KUKA KRL program: MyProgram_167().src

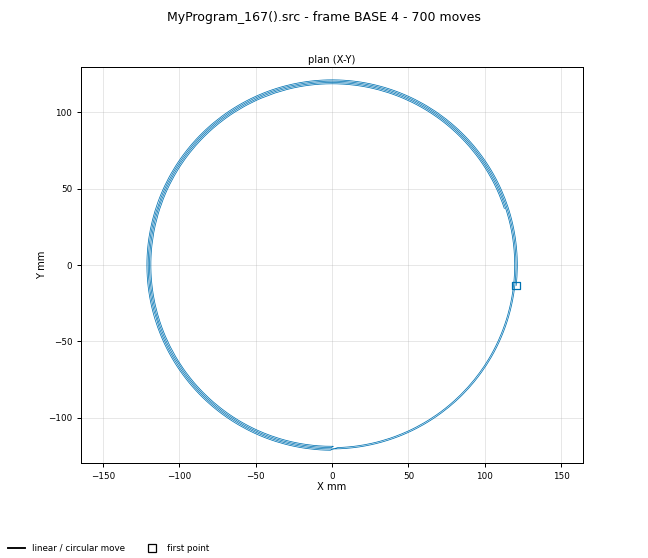
[picture p0: tool path of MyProgram_167().src in frame BASE 4, 700 of 700 moves have a stored position in this frame; points joined in program order, loops and branches not executed]
&ACCESS RVP
&REL 1
&PARAM TEMPLATE = C:\KRC\Roboter\Template\vorgabe
&PARAM EDITMASK = *
DEF MyProgram_167()
; ---- Setting reference (Base) ----
$BASE = BASE_DATA[4]

; --------------------------
; ---- Setting tool (TCP) ----
$TOOL = TOOL_DATA[3]
; --------------------------

$VEL.CP = VEL_APROX_PRINT
Startdeposition()
$VEL.CP = VEL_PRINT
LIN {X 120.5088,Y -13.3642,Z 126,A -9.8164,B 24.9507,C -1.6218,E1 25.1589,E2 455.9216} C_DIS
LIN {X 120.8004,Y -10.4027,Z 126,A -8.4201,B 24.9505,C -1.6259,E1 25.1593,E2 454.5239} C_DIS
LIN {X 121.0193,Y -7.435,Z 126,A -7.0235,B 24.9502,C -1.63,E1 25.1595,E2 453.1259} C_DIS
LIN {X 121.1789,Y -4.022,Z 126,A -5.6063,B 24.9505,C -1.6254,E1 25.1597,E2 451.728} C_DIS
LIN {X 121.2384,Y -1.4879,Z 126,A -4.2539,B 24.9498,C -1.6371,E1 25.1597,E2 450.3561} C_DIS
LIN {X 121.2384,Y 1.4879,Z 126,A -2.834,B 24.9495,C -1.6424,E1 25.1597,E2 448.9323} C_DIS
LIN {X 121.1654,Y 4.4628,Z 126,A -1.4376,B 24.9492,C -1.6465,E1 25.1597,E2 447.5345} C_DIS
LIN {X 121.0193,Y 7.435,Z 126,A -0.0409,B 24.9489,C -1.6506,E1 25.1594,E2 446.1364} C_DIS
LIN {X 120.7573,Y 10.8703,Z 126,A 1.6055,B 24.9486,C -1.6568,E1 25.159,E2 444.4851} C_DIS
LIN {X 120.3357,Y 14.842,Z 126,A 3.4507,B 24.9483,C -1.6607,E1 25.1585,E2 442.6415} C_DIS
LIN {X 119.9352,Y 17.7907,Z 126,A 4.8473,B 24.9481,C -1.6648,E1 25.1579,E2 441.2437} C_DIS
LIN {X 119.4625,Y 20.7287,Z 126,A 6.2442,B 24.9478,C -1.6688,E1 25.1573,E2 439.8455} C_DIS
LIN {X 118.9178,Y 23.6542,Z 126,A 7.6407,B 24.9476,C -1.6728,E1 25.1565,E2 438.4477} C_DIS
LIN {X 118.3015,Y 26.5655,Z 126,A 9.0377,B 24.9473,C -1.6767,E1 25.1557,E2 437.0495} C_DIS
LIN {X 117.6139,Y 29.4607,Z 126,A 10.4346,B 24.9471,C -1.6807,E1 25.1548,E2 435.6514} C_DIS
LIN {X 116.8555,Y 32.3383,Z 126,A 11.8317,B 24.9468,C -1.6846,E1 25.1537,E2 434.2532} C_DIS
LIN {X 116.0266,Y 35.1963,Z 126,A 13.2287,B 24.9466,C -1.6884,E1 25.1526,E2 432.855} C_DIS
LIN {X 115.1279,Y 38.0331,Z 126,A 14.6257,B 24.9463,C -1.6923,E1 25.1514,E2 431.4568} C_DIS
LIN {X 114.0244,Y 41.2185,Z 126,A 16.0417,B 24.9466,C -1.6883,E1 25.1501,E2 430.0583} C_DIS
LIN {X 113.1231,Y 43.6364,Z 126,A 17.5207,B 24.9455,C -1.7048,E1 25.1486,E2 428.5485} C_DIS
LIN {X 111.7931,Y 46.9333,Z 126,A 18.8451,B 24.9463,C -1.6921,E1 25.1473,E2 427.2613} C_DIS
LIN {X 110.8457,Y 49.1345,Z 126,A 20.2154,B 24.9454,C -1.7072,E1 25.1457,E2 425.863} C_DIS
LIN {X 109.6065,Y 51.84,Z 126,A 21.613,B 24.9451,C -1.7108,E1 25.1441,E2 424.4644} C_DIS
LIN {X 108.3012,Y 54.5143,Z 126,A 23.0108,B 24.9449,C -1.7144,E1 25.1423,E2 423.0656} C_DIS
LIN {X 106.9308,Y 57.1557,Z 126,A 24.4089,B 24.9447,C -1.7179,E1 25.1405,E2 421.6666} C_DIS
LIN {X 105.4959,Y 59.7627,Z 126,A 25.9523,B 24.944,C -1.7286,E1 25.1384,E2 420.106} C_DIS
LIN {X 103.9975,Y 62.3337,Z 126,A 27.2051,B 24.9442,C -1.7248,E1 25.1366,E2 418.8687} C_DIS
LIN {X 102.4364,Y 64.8671,Z 126,A 28.6034,B 24.944,C -1.7281,E1 25.1345,E2 417.4696} C_DIS
LIN {X 100.8136,Y 67.3615,Z 126,A 30.1196,B 24.9434,C -1.7372,E1 25.1322,E2 415.9394} C_DIS
LIN {X 98.2659,Y 71.0265,Z 126,A 32.0998,B 24.9435,C -1.7363,E1 25.129,E2 413.9712} C_DIS
LIN {X 96.4932,Y 73.4167,Z 126,A 33.4984,B 24.9433,C -1.7394,E1 25.1267,E2 412.5719} C_DIS
LIN {X 94.6625,Y 75.7627,Z 126,A 34.8975,B 24.9431,C -1.7425,E1 25.1242,E2 411.172} C_DIS
LIN {X 92.7746,Y 78.063,Z 126,A 36.2965,B 24.9429,C -1.7455,E1 25.1217,E2 409.7723} C_DIS
LIN {X 90.8309,Y 80.3163,Z 126,A 37.6959,B 24.9427,C -1.7484,E1 25.1192,E2 408.3724} C_DIS
LIN {X 88.8325,Y 82.5212,Z 126,A 39.0953,B 24.9425,C -1.7513,E1 25.1165,E2 406.9724} C_DIS
LIN {X 86.7806,Y 84.6764,Z 126,A 40.4951,B 24.9423,C -1.7541,E1 25.1138,E2 405.572} C_DIS
LIN {X 84.6764,Y 86.7806,Z 126,A 41.8949,B 24.9422,C -1.7568,E1 25.111,E2 404.1717} C_DIS
LIN {X 82.5212,Y 88.8325,Z 126,A 43.2949,B 24.942,C -1.7594,E1 25.1082,E2 402.7712} C_DIS
LIN {X 80.3163,Y 90.8309,Z 126,A 44.8186,B 24.9414,C -1.768,E1 25.105,E2 401.2334} C_DIS
LIN {X 77.6174,Y 93.1449,Z 126,A 46.368,B 24.9416,C -1.7649,E1 25.1017,E2 399.6971} C_DIS
LIN {X 74.5953,Y 95.585,Z 126,A 48.1962,B 24.9414,C -1.768,E1 25.0977,E2 397.8685} C_DIS
LIN {X 72.0735,Y 97.4993,Z 126,A 49.6061,B 24.9415,C -1.7665,E1 25.0946,E2 396.4672} C_DIS
LIN {X 69.8153,Y 99.1301,Z 126,A 50.9982,B 24.9411,C -1.7725,E1 25.0914,E2 395.0659} C_DIS
LIN {X 67.3615,Y 100.8136,Z 126,A 52.3996,B 24.941,C -1.7746,E1 25.0881,E2 393.6643} C_DIS
LIN {X 64.7375,Y 102.5174,Z 126,A 53.8079,B 24.941,C -1.7736,E1 25.0849,E2 392.2629} C_DIS
LIN {X 62.3337,Y 103.9975,Z 126,A 55.2026,B 24.9407,C -1.7785,E1 25.0815,E2 390.8609} C_DIS
LIN {X 59.7627,Y 105.4959,Z 126,A 56.6046,B 24.9406,C -1.7804,E1 25.0781,E2 389.4587} C_DIS
LIN {X 56.9784,Y 107.0241,Z 126,A 58.0159,B 24.9407,C -1.7782,E1 25.0747,E2 388.0567} C_DIS
LIN {X 54.5143,Y 108.3012,Z 126,A 59.409,B 24.9404,C -1.7838,E1 25.0712,E2 386.6541} C_DIS
LIN {X 51.84,Y 109.6065,Z 126,A 60.8116,B 24.9403,C -1.7853,E1 25.0676,E2 385.2515} C_DIS
LIN {X 48.6786,Y 111.0444,Z 126,A 62.4707,B 24.9401,C -1.7881,E1 25.0634,E2 383.59} C_DIS
LIN {X 45.0213,Y 112.5791,Z 126,A 64.3189,B 24.9401,C -1.7888,E1 25.0586,E2 381.7443} C_DIS
LIN {X 42.2449,Y 113.65,Z 126,A 65.7222,B 24.9399,C -1.79,E1 25.055,E2 380.3412} C_DIS
LIN {X 39.4431,Y 114.6525,Z 126,A 67.1257,B 24.9399,C -1.7912,E1 25.0513,E2 378.9378} C_DIS
LIN {X 36.6175,Y 115.586,Z 126,A 68.5295,B 24.9398,C -1.7922,E1 25.0476,E2 377.5342} C_DIS
LIN {X 33.7698,Y 116.4498,Z 126,A 69.9336,B 24.9398,C -1.7931,E1 25.0438,E2 376.1303} C_DIS
LIN {X 30.9018,Y 117.2435,Z 126,A 71.3378,B 24.9397,C -1.794,E1 25.04,E2 374.7263} C_DIS
LIN {X 28.0152,Y 117.9666,Z 126,A 72.7421,B 24.9397,C -1.7947,E1 25.0362,E2 373.3224} C_DIS
LIN {X 25.1117,Y 118.6186,Z 126,A 74.1469,B 24.9396,C -1.7953,E1 25.0324,E2 371.9178} C_DIS
LIN {X 22.1931,Y 119.1991,Z 126,A 75.7244,B 24.939,C -1.804,E1 25.028,E2 370.3218} C_DIS
LIN {X 19.2612,Y 119.7078,Z 126,A 76.9573,B 24.9395,C -1.7963,E1 25.0246,E2 369.1082} C_DIS
LIN {X 16.3176,Y 120.1445,Z 126,A 78.3627,B 24.9395,C -1.7967,E1 25.0208,E2 367.7033} C_DIS
LIN {X 13.3642,Y 120.5088,Z 126,A 79.7685,B 24.9395,C -1.7969,E1 25.0169,E2 366.298} C_DIS
LIN {X 10.4027,Y 120.8004,Z 126,A 81.1742,B 24.9395,C -1.797,E1 25.013,E2 364.8928} C_DIS
LIN {X 7.435,Y 121.0193,Z 126,A 82.5805,B 24.9395,C -1.797,E1 25.009,E2 363.4871} C_DIS
LIN {X 4.4628,Y 121.1654,Z 126,A 84.1576,B 24.9389,C -1.8049,E1 25.0046,E2 361.8918} C_DIS
LIN {X 0.8202,Y 121.2425,Z 126,A 85.687,B 24.9396,C -1.7958,E1 25.0004,E2 360.3842} C_DIS
LIN {X -2.9756,Y 121.211,Z 126,A 87.5041,B 24.9396,C -1.7964,E1 24.9953,E2 358.5656} C_DIS
LIN {X -5.9493,Y 121.1015,Z 126,A 88.9114,B 24.9396,C -1.7959,E1 24.9914,E2 357.159} C_DIS
LIN {X -8.9195,Y 120.919,Z 126,A 90.319,B 24.9396,C -1.7954,E1 24.9875,E2 355.7522} C_DIS
LIN {X -11.8843,Y 120.6637,Z 126,A 91.7265,B 24.9396,C -1.7948,E1 24.9835,E2 354.3454} C_DIS
LIN {X -14.842,Y 120.3357,Z 126,A 93.1491,B 24.9396,C -1.7948,E1 24.9796,E2 352.9221} C_DIS
LIN {X -17.7907,Y 119.9352,Z 126,A 94.5427,B 24.9397,C -1.7932,E1 24.9758,E2 351.5309} C_DIS
LIN {X -20.7287,Y 119.4625,Z 126,A 95.9513,B 24.9397,C -1.7923,E1 24.9719,E2 350.1231} C_DIS
LIN {X -23.6542,Y 118.9178,Z 126,A 97.3599,B 24.9399,C -1.7913,E1 24.968,E2 348.7153} C_DIS
LIN {X -26.5655,Y 118.3015,Z 126,A 98.9351,B 24.9394,C -1.7977,E1 24.9637,E2 347.123} C_DIS
LIN {X -30.9018,Y 117.2435,Z 126,A 100.8828,B 24.9401,C -1.7883,E1 24.9585,E2 345.1949} C_DIS
LIN {X -33.7698,Y 116.4498,Z 126,A 102.2921,B 24.9401,C -1.7869,E1 24.9547,E2 343.7865} C_DIS
LIN {X -36.6175,Y 115.586,Z 126,A 103.7017,B 24.9403,C -1.7854,E1 24.9509,E2 342.378} C_DIS
LIN {X -39.4431,Y 114.6525,Z 126,A 105.1119,B 24.9403,C -1.7839,E1 24.9472,E2 340.9688} C_DIS
LIN {X -42.2449,Y 113.65,Z 126,A 106.5502,B 24.9403,C -1.7835,E1 24.9434,E2 339.5285} C_DIS
LIN {X -45.0213,Y 112.5791,Z 126,A 107.9324,B 24.9406,C -1.7805,E1 24.9398,E2 338.1506} C_DIS
LIN {X -47.7706,Y 111.4403,Z 126,A 109.3428,B 24.9407,C -1.7786,E1 24.9362,E2 336.7413} C_DIS
LIN {X -50.4911,Y 110.2344,Z 126,A 110.7536,B 24.9408,C -1.7767,E1 24.9326,E2 335.3316} C_DIS
LIN {X -53.1811,Y 108.9621,Z 126,A 112.1649,B 24.941,C -1.7747,E1 24.9291,E2 333.9215} C_DIS
LIN {X -55.8619,Y 107.6121,Z 126,A 113.7461,B 24.9406,C -1.7796,E1 24.9251,E2 332.3244} C_DIS
LIN {X -58.9695,Y 105.9388,Z 126,A 115.2623,B 24.9413,C -1.77,E1 24.9214,E2 330.8267} C_DIS
LIN {X -62.3337,Y 103.9975,Z 126,A 117.1167,B 24.9415,C -1.7674,E1 24.917,E2 328.9728} C_DIS
LIN {X -64.8671,Y 102.4364,Z 126,A 118.5171,B 24.9416,C -1.7645,E1 24.9137,E2 327.5749} C_DIS
LIN {X -67.3615,Y 100.8136,Z 126,A 119.9293,B 24.9418,C -1.762,E1 24.9104,E2 326.164} C_DIS
LIN {X -69.8153,Y 99.1301,Z 126,A 121.3416,B 24.942,C -1.7594,E1 24.9071,E2 324.753} C_DIS
LIN {X -72.2271,Y 97.3869,Z 126,A 122.7544,B 24.9422,C -1.7568,E1 24.9039,E2 323.3415} C_DIS
LIN {X -75.0019,Y 95.2637,Z 126,A 124.1911,B 24.943,C -1.7438,E1 24.9008,E2 321.9303} C_DIS
LIN {X -76.9186,Y 93.7256,Z 126,A 125.5798,B 24.9425,C -1.7512,E1 24.8978,E2 320.5189} C_DIS
LIN {X -79.1956,Y 91.8097,Z 126,A 126.9929,B 24.9427,C -1.7483,E1 24.8948,E2 319.1072} C_DIS
LIN {X -81.4249,Y 89.8385,Z 126,A 128.4063,B 24.9429,C -1.7454,E1 24.8918,E2 317.6951} C_DIS
LIN {X -83.6051,Y 87.8132,Z 126,A 129.9755,B 24.9427,C -1.7492,E1 24.8886,E2 316.1105} C_DIS
LIN {X -86.8025,Y 84.6536,Z 126,A 131.9416,B 24.9435,C -1.737,E1 24.8848,E2 314.1649} C_DIS
LIN {X -88.8325,Y 82.5212,Z 126,A 133.3537,B 24.9436,C -1.7344,E1 24.8821,E2 312.7528} C_DIS
LIN {X -90.8309,Y 80.3163,Z 126,A 134.768,B 24.9438,C -1.7312,E1 24.8794,E2 311.34} C_DIS
LIN {X -92.7964,Y 78.0368,Z 126,A 136.1837,B 24.9441,C -1.7272,E1 24.8769,E2 309.9273} C_DIS
LIN {X -94.9311,Y 75.4227,Z 126,A 137.8426,B 24.9441,C -1.7258,E1 24.874,E2 308.2641} C_DIS
LIN {X -97.3869,Y 72.2271,Z 126,A 139.7182,B 24.9446,C -1.7193,E1 24.8708,E2 306.3951} C_DIS
LIN {X -99.1301,Y 69.8153,Z 126,A 141.1328,B 24.9448,C -1.7157,E1 24.8685,E2 304.9819} C_DIS
LIN {X -100.8136,Y 67.3615,Z 126,A 142.5475,B 24.9451,C -1.7121,E1 24.8663,E2 303.5687} C_DIS
LIN {X -102.4364,Y 64.8671,Z 126,A 143.9623,B 24.9453,C -1.7085,E1 24.8642,E2 302.1554} C_DIS
LIN {X -104.1525,Y 62.0714,Z 126,A 145.3916,B 24.9459,C -1.6988,E1 24.8621,E2 300.7419} C_DIS
LIN {X -105.4959,Y 59.7627,Z 126,A 146.7923,B 24.9458,C -1.7011,E1 24.8602,E2 299.3285} C_DIS
LIN {X -106.9308,Y 57.1557,Z 126,A 148.2076,B 24.946,C -1.6973,E1 24.8583,E2 297.9147} C_DIS
LIN {X -108.3095,Y 54.4976,Z 126,A 149.6237,B 24.9463,C -1.6931,E1 24.8565,E2 296.501} C_DIS
LIN {X -109.6065,Y 51.84,Z 126,A 151.0383,B 24.9465,C -1.6896,E1 24.8548,E2 295.0871} C_DIS
LIN {X -110.8457,Y 49.1345,Z 126,A 152.4539,B 24.9467,C -1.6857,E1 24.8532,E2 293.6731} C_DIS
LIN {X -112.0181,Y 46.3994,Z 126,A 153.8695,B 24.947,C -1.6818,E1 24.8516,E2 292.259} C_DIS
LIN {X -113.1231,Y 43.6364,Z 126,A 155.2851,B 24.9472,C -1.6778,E1 24.8502,E2 290.8449} C_DIS
LIN {X -114.1599,Y 40.8471,Z 126,A 156.7007,B 24.9475,C -1.6738,E1 24.8488,E2 289.4308} C_DIS
LIN {X -115.2699,Y 37.5944,Z 126,A 158.1384,B 24.9483,C -1.6607,E1 24.8476,E2 288.0162} C_DIS
LIN {X -116.0266,Y 35.1963,Z 126,A 159.6235,B 24.9478,C -1.6696,E1 24.8463,E2 286.5012} C_DIS
LIN {X -117.0066,Y 31.7789,Z 126,A 160.9754,B 24.949,C -1.6502,E1 24.8453,E2 285.1878} C_DIS
LIN {X -117.6139,Y 29.4607,Z 126,A 162.4636,B 24.9483,C -1.6618,E1 24.8443,E2 283.6633} C_DIS
LIN {X -118.4249,Y 25.9994,Z 126,A 163.8076,B 24.9495,C -1.642,E1 24.8435,E2 282.3586} C_DIS
LIN {X -118.9626,Y 23.4216,Z 126,A 165.2076,B 24.9493,C -1.6446,E1 24.8427,E2 280.9441} C_DIS
LIN {X -119.4625,Y 20.7287,Z 126,A 166.6128,B 24.9493,C -1.6451,E1 24.842,E2 279.5293} C_DIS
LIN {X -119.9352,Y 17.7907,Z 126,A 168.0287,B 24.9495,C -1.641,E1 24.8414,E2 278.1149} C_DIS
LIN {X -120.3357,Y 14.842,Z 126,A 169.4448,B 24.9498,C -1.6368,E1 24.8409,E2 276.7003} C_DIS
LIN {X -120.6637,Y 11.8843,Z 126,A 170.8611,B 24.9501,C -1.6327,E1 24.8405,E2 275.2854} C_DIS
LIN {X -120.919,Y 8.9195,Z 126,A 172.2771,B 24.9503,C -1.6285,E1 24.8401,E2 273.8708} C_DIS
LIN {X -121.1015,Y 5.9493,Z 126,A 173.6934,B 24.9506,C -1.6243,E1 24.8399,E2 272.4559} C_DIS
LIN {X -121.211,Y 2.9756,Z 126,A 175.1095,B 24.9508,C -1.6201,E1 24.8399,E2 271.0413} C_DIS
LIN {X -121.2455,Y -0.4051,Z 126,A 176.7824,B 24.9509,C -1.6182,E1 24.8398,E2 269.3629} C_DIS
LIN {X -121.1654,Y -4.4628,Z 126,A 178.6495,B 24.9514,C -1.6097,E1 24.8399,E2 267.5048} C_DIS
LIN {X -121.013,Y -7.5284,Z 126,A -179.7941,B 24.9514,C -1.6097,E1 24.8402,E2 265.9393} C_DIS
LIN {X -120.6637,Y -11.8843,Z 126,A -177.8103,B 24.9521,C -1.5994,E1 24.8407,E2 263.9679} C_DIS
LIN {X -120.3357,Y -14.842,Z 126,A -176.3942,B 24.9523,C -1.5953,E1 24.8411,E2 262.5531} C_DIS
LIN {X -119.9352,Y -17.7907,Z 126,A -174.9784,B 24.9526,C -1.5912,E1 24.8417,E2 261.1386} C_DIS
LIN {X -119.4625,Y -20.7287,Z 126,A -173.5624,B 24.9528,C -1.5872,E1 24.8423,E2 259.7238} C_DIS
LIN {X -118.9178,Y -23.6542,Z 126,A -172.1466,B 24.953,C -1.5831,E1 24.8431,E2 258.3092} C_DIS
LIN {X -118.3015,Y -26.5655,Z 126,A -170.7307,B 24.9533,C -1.5791,E1 24.8439,E2 256.8945} C_DIS
LIN {X -117.6139,Y -29.4607,Z 126,A -169.3152,B 24.9535,C -1.5752,E1 24.8449,E2 255.4803} C_DIS
LIN {X -116.8555,Y -32.3383,Z 126,A -167.8998,B 24.9537,C -1.5712,E1 24.8459,E2 254.0661} C_DIS
LIN {X -116.0266,Y -35.1963,Z 126,A -166.4841,B 24.954,C -1.5673,E1 24.847,E2 252.6515} C_DIS
LIN {X -115.0484,Y -38.2691,Z 126,A -164.8855,B 24.954,C -1.5659,E1 24.8484,E2 251.047} C_DIS
LIN {X -114.1599,Y -40.8471,Z 126,A -163.6533,B 24.9544,C -1.5596,E1 24.8496,E2 249.823} C_DIS
LIN {X -113.0904,Y -43.7196,Z 126,A -162.2341,B 24.9548,C -1.554,E1 24.8509,E2 248.409} C_DIS
LIN {X -112.0181,Y -46.3994,Z 126,A -160.8227,B 24.9548,C -1.5521,E1 24.8524,E2 246.9945} C_DIS
LIN {X -110.8457,Y -49.1345,Z 126,A -159.4081,B 24.9551,C -1.5483,E1 24.854,E2 245.5809} C_DIS
LIN {X -109.6065,Y -51.84,Z 126,A -157.993,B 24.9553,C -1.5447,E1 24.8557,E2 244.1668} C_DIS
LIN {X -108.3012,Y -54.5143,Z 126,A -156.5784,B 24.9555,C -1.5411,E1 24.8574,E2 242.7531} C_DIS
LIN {X -106.9308,Y -57.1557,Z 126,A -155.1021,B 24.9555,C -1.5402,E1 24.8594,E2 241.271} C_DIS
LIN {X -105.2072,Y -60.2651,Z 126,A -153.4738,B 24.9559,C -1.5334,E1 24.8616,E2 239.6504} C_DIS
LIN {X -103.2247,Y -63.6052,Z 126,A -151.6275,B 24.9562,C -1.5289,E1 24.8643,E2 237.8053} C_DIS
LIN {X -101.6327,Y -66.1193,Z 126,A -150.2134,B 24.9564,C -1.5256,E1 24.8664,E2 236.3921} C_DIS
LIN {X -99.8332,Y -68.8039,Z 126,A -148.5835,B 24.9564,C -1.5262,E1 24.869,E2 234.7526} C_DIS
LIN {X -97.9236,Y -71.494,Z 126,A -147.1102,B 24.9568,C -1.5185,E1 24.8713,E2 233.2904} C_DIS
LIN {X -95.5851,Y -74.5953,Z 126,A -145.2649,B 24.957,C -1.5144,E1 24.8745,E2 231.4462} C_DIS
LIN {X -93.7256,Y -76.9186,Z 126,A -143.8516,B 24.9572,C -1.5113,E1 24.877,E2 230.0335} C_DIS
LIN {X -91.8097,Y -79.1956,Z 126,A -142.4382,B 24.9574,C -1.5084,E1 24.8795,E2 228.6208} C_DIS
LIN {X -89.8385,Y -81.4249,Z 126,A -140.9105,B 24.9573,C -1.5106,E1 24.8824,E2 227.081} C_DIS
LIN {X -86.7806,Y -84.6764,Z 126,A -138.9054,B 24.9578,C -1.5013,E1 24.8862,E2 225.0894} C_DIS
LIN {X -84.6764,Y -86.7806,Z 126,A -137.4929,B 24.9579,C -1.4985,E1 24.889,E2 223.6774} C_DIS
LIN {X -82.5212,Y -88.8325,Z 126,A -135.9178,B 24.9577,C -1.5032,E1 24.8923,E2 222.0848} C_DIS
LIN {X -80.3163,Y -90.8309,Z 126,A -134.6681,B 24.9582,C -1.4933,E1 24.8949,E2 220.8536} C_DIS
LIN {X -78.063,Y -92.7746,Z 126,A -133.2263,B 24.9582,C -1.4922,E1 24.8979,E2 219.4088} C_DIS
LIN {X -75.7627,Y -94.6625,Z 126,A -131.7323,B 24.9582,C -1.4935,E1 24.9012,E2 217.9062} C_DIS
LIN {X -73.4167,Y -96.4932,Z 126,A -130.4327,B 24.9586,C -1.4862,E1 24.904,E2 216.6193} C_DIS
LIN {X -71.0265,Y -98.2659,Z 126,A -129.0209,B 24.9587,C -1.484,E1 24.9072,E2 215.2078} C_DIS
LIN {X -68.5936,Y -99.9794,Z 126,A -127.5133,B 24.9587,C -1.4862,E1 24.9107,E2 213.6898} C_DIS
LIN {X -66.1193,Y -101.6327,Z 126,A -126.1986,B 24.959,C -1.4798,E1 24.9137,E2 212.3859} C_DIS
LIN {X -63.6052,Y -103.2247,Z 126,A -124.7876,B 24.959,C -1.4778,E1 24.9171,E2 210.9752} C_DIS
LIN {X -61.0528,Y -104.7546,Z 126,A -123.2908,B 24.959,C -1.4799,E1 24.9207,E2 209.4689} C_DIS
LIN {X -57.9543,Y -106.4976,Z 126,A -121.9393,B 24.9599,C -1.4627,E1 24.9239,E2 208.1545} C_DIS
LIN {X -55.8392,Y -107.6241,Z 126,A -120.4877,B 24.9592,C -1.4757,E1 24.9276,E2 206.6679} C_DIS
LIN {X -53.1811,Y -108.9621,Z 126,A -118.9981,B 24.9591,C -1.4777,E1 24.9313,E2 205.1695} C_DIS
LIN {X -50.4911,Y -110.2344,Z 126,A -117.7365,B 24.9595,C -1.4695,E1 24.9345,E2 203.9244} C_DIS
LIN {X -47.7706,Y -111.4403,Z 126,A -116.3273,B 24.9596,C -1.4681,E1 24.9381,E2 202.5153} C_DIS
LIN {X -45.0213,Y -112.5791,Z 126,A -114.9176,B 24.9596,C -1.4668,E1 24.9418,E2 201.1055} C_DIS
LIN {X -42.2449,Y -113.65,Z 126,A -113.5087,B 24.9598,C -1.4656,E1 24.9454,E2 199.6964} C_DIS
LIN {X -39.4431,Y -114.6525,Z 126,A -112.0997,B 24.9598,C -1.4645,E1 24.9491,E2 198.2873} C_DIS
LIN {X -36.6175,Y -115.586,Z 126,A -110.6913,B 24.9598,C -1.4635,E1 24.9529,E2 196.8787} C_DIS
LIN {X -33.4991,Y -116.5265,Z 126,A -109.0639,B 24.9598,C -1.4665,E1 24.9573,E2 195.2415} C_DIS
LIN {X -30.9018,Y -117.2435,Z 126,A -107.8747,B 24.96,C -1.4618,E1 24.9605,E2 194.0616} C_DIS
LIN {X -28.0152,Y -117.9666,Z 126,A -106.4671,B 24.96,C -1.4611,E1 24.9643,E2 192.6537} C_DIS
LIN {X -25.1117,Y -118.6186,Z 126,A -105.0151,B 24.96,C -1.4626,E1 24.9683,E2 191.1965} C_DIS
LIN {X -22.1931,Y -119.1991,Z 126,A -103.6519,B 24.96,C -1.46,E1 24.972,E2 189.8378} C_DIS
LIN {X -19.2612,Y -119.7078,Z 126,A -102.2445,B 24.96,C -1.4596,E1 24.9759,E2 188.43} C_DIS
LIN {X -16.3176,Y -120.1445,Z 126,A -100.8377,B 24.9601,C -1.4593,E1 24.9798,E2 187.0228} C_DIS
LIN {X -12.8412,Y -120.5635,Z 126,A -99.3639,B 24.9606,C -1.4507,E1 24.9838,E2 185.5686} C_DIS
LIN {X -10.4027,Y -120.8004,Z 126,A -98.0247,B 24.9601,C -1.4591,E1 24.9876,E2 184.2088} C_DIS
LIN {X -7.435,Y -121.0193,Z 126,A -96.6184,B 24.9601,C -1.4591,E1 24.9915,E2 182.8019} C_DIS
LIN {X -4.4628,Y -121.1654,Z 126,A -95.2124,B 24.9601,C -1.4592,E1 24.9954,E2 181.3953} C_DIS
LIN {X -1.1524,Y -121.2404,Z 126,A -93.5793,B 24.9599,C -1.4627,E1 25,E2 179.7537} C_DIS
LIN {X -1.1524,Y -121.2404,Z 126,A -93.5793,B 24.9599,C -1.4627,E1 25,E2 179.7537} C_DIS
Enddeposition()
LIN {X 0.8412,Y -120.3739,Z 126,A -92.3537,B 24.9583,C -1.4914,E1 25.0036,E2 178.4603} C_DIS
Startdeposition()
$VEL.CP = VEL_PRINT
LIN {X -0.5989,Y -120.3841,Z 126,A -94.8852,B 24.963,C -1.4054,E1 24.996,E2 181.1955} C_DIS
LIN {X -6.0161,Y -120.2368,Z 126,A -96.5858,B 24.9609,C -1.4454,E1 24.9915,E2 182.8019} C_DIS
LIN {X -10.8702,Y -119.8939,Z 126,A -98.8361,B 24.9607,C -1.4484,E1 24.9853,E2 185.0458} C_DIS
LIN {X -17.8185,Y -119.061,Z 126,A -102.2139,B 24.9607,C -1.4467,E1 24.9759,E2 188.43} C_DIS
LIN {X -20.8825,Y -118.5613,Z 126,A -103.8801,B 24.9612,C -1.4386,E1 24.9712,E2 190.1171} C_DIS
LIN {X -24.3819,Y -117.8908,Z 126,A -105.4909,B 24.961,C -1.4432,E1 24.9668,E2 191.7189} C_DIS
LIN {X -27.3946,Y -117.2276,Z 126,A -106.9794,B 24.961,C -1.443,E1 24.9628,E2 193.2097} C_DIS
LIN {X -31.3064,Y -116.2437,Z 126,A -108.9016,B 24.961,C -1.444,E1 24.9576,E2 195.1323} C_DIS
LIN {X -34.7415,Y -115.2648,Z 126,A -110.6525,B 24.961,C -1.4429,E1 24.9529,E2 196.8888} C_DIS
LIN {X -38.9685,Y -113.9053,Z 126,A -112.6607,B 24.9607,C -1.4493,E1 24.9476,E2 198.8854} C_DIS
LIN {X -41.7005,Y -112.9335,Z 126,A -114.0929,B 24.9607,C -1.4482,E1 24.9438,E2 200.3231} C_DIS
LIN {X -44.8377,Y -111.7256,Z 126,A -115.7945,B 24.9609,C -1.4452,E1 24.9393,E2 202.0355} C_DIS
LIN {X -50.3958,Y -109.3304,Z 126,A -118.4173,B 24.9601,C -1.4599,E1 24.9327,E2 204.6295} C_DIS
LIN {X -54.199,Y -107.4965,Z 126,A -120.6944,B 24.9606,C -1.4504,E1 24.9269,E2 206.9351} C_DIS
LIN {X -57.631,Y -105.6949,Z 126,A -122.5226,B 24.9604,C -1.4537,E1 24.9224,E2 208.7608} C_DIS
LIN {X -61.1673,Y -103.6882,Z 126,A -124.4381,B 24.9602,C -1.4573,E1 24.9178,E2 210.6733} C_DIS
LIN {X -66.0537,Y -100.6461,Z 126,A -127.2092,B 24.9601,C -1.4602,E1 24.9113,E2 213.4465} C_DIS
LIN {X -69.5283,Y -98.2788,Z 126,A -129.3194,B 24.9601,C -1.4587,E1 24.9064,E2 215.5674} C_DIS
LIN {X -72.3405,Y -96.2265,Z 126,A -130.8139,B 24.9596,C -1.4688,E1 24.9031,E2 217.0432} C_DIS
LIN {X -75.431,Y -93.8247,Z 126,A -132.7809,B 24.9596,C -1.4676,E1 24.8988,E2 219.0202} C_DIS
LIN {X -78.3202,Y -91.4261,Z 126,A -134.5227,B 24.9593,C -1.4731,E1 24.8951,E2 220.7557} C_DIS
LIN {X -81.8326,Y -88.2975,Z 126,A -136.8819,B 24.9593,C -1.4723,E1 24.8902,E2 223.1262} C_DIS
LIN {X -84.6892,Y -85.5595,Z 126,A -138.6133,B 24.9588,C -1.483,E1 24.8867,E2 224.8395} C_DIS
LIN {X -87.0575,Y -83.1502,Z 126,A -140.4053,B 24.959,C -1.4785,E1 24.8832,E2 226.6499} C_DIS
LIN {X -90.0389,Y -79.9121,Z 126,A -142.3047,B 24.9583,C -1.4917,E1 24.8797,E2 228.5263} C_DIS
LIN {X -91.9932,Y -77.6545,Z 126,A -143.6954,B 24.9581,C -1.4963,E1 24.8772,E2 229.9123} C_DIS
LIN {X -93.842,Y -75.4095,Z 126,A -145.1049,B 24.9579,C -1.4986,E1 24.8747,E2 231.3231} C_DIS
LIN {X -95.9831,Y -72.6644,Z 126,A -146.9284,B 24.9581,C -1.4954,E1 24.8716,E2 233.1627} C_DIS
LIN {X -98.1563,Y -69.7,Z 126,A -148.5818,B 24.9576,C -1.504,E1 24.8689,E2 234.8038} C_DIS
LIN {X -100.3223,Y -66.5448,Z 126,A -150.8614,B 24.9585,C -1.4891,E1 24.8653,E2 237.1302} C_DIS
LIN {X -102.3672,Y -63.3552,Z 126,A -152.1202,B 24.9569,C -1.5171,E1 24.8635,E2 238.3287} C_DIS
LIN {X -103.6927,Y -61.1598,Z 126,A -153.4838,B 24.957,C -1.5143,E1 24.8615,E2 239.7061} C_DIS
LIN {X -105.8961,Y -57.2602,Z 126,A -155.5468,B 24.9565,C -1.5231,E1 24.8587,E2 241.759} C_DIS
LIN {X -107.3144,Y -54.5561,Z 126,A -157.0698,B 24.9565,C -1.5242,E1 24.8568,E2 243.2876} C_DIS
LIN {X -108.8327,Y -51.4636,Z 126,A -158.845,B 24.9565,C -1.523,E1 24.8546,E2 245.0751} C_DIS
LIN {X -110.7819,Y -47.1191,Z 126,A -161.0288,B 24.956,C -1.5331,E1 24.8522,E2 247.2468} C_DIS
LIN {X -112.0412,Y -44.0393,Z 126,A -162.6061,B 24.9557,C -1.5381,E1 24.8505,E2 248.8212} C_DIS
LIN {X -113.3257,Y -40.6251,Z 126,A -164.665,B 24.9562,C -1.5296,E1 24.8485,E2 250.9119} C_DIS
LIN {X -116.504,Y -30.3254,Z 126,A -169.6309,B 24.9549,C -1.5523,E1 24.8446,E2 255.8525} C_DIS
LIN {X -117.4548,Y -26.4109,Z 126,A -171.3796,B 24.9541,C -1.5654,E1 24.8435,E2 257.5801} C_DIS
LIN {X -118.1445,Y -23.1231,Z 126,A -173.0283,B 24.9539,C -1.5683,E1 24.8426,E2 259.2316} C_DIS
LIN {X -118.8059,Y -19.4424,Z 126,A -174.8009,B 24.9536,C -1.5743,E1 24.8417,E2 261.0005} C_DIS
LIN {X -119.323,Y -15.9668,Z 126,A -176.5395,B 24.9534,C -1.5768,E1 24.8411,E2 262.7433} C_DIS
LIN {X -119.7529,Y -12.327,Z 126,A -178.3277,B 24.9532,C -1.5806,E1 24.8405,E2 264.5332} C_DIS
LIN {X -120.0944,Y -8.3705,Z 126,A 179.8324,B 24.9527,C -1.5888,E1 24.8401,E2 266.3646} C_DIS
LIN {X -120.2932,Y -4.7339,Z 126,A 178.1733,B 24.9522,C -1.5976,E1 24.8399,E2 268.0128} C_DIS
LIN {X -120.3698,Y -1.9603,Z 126,A 176.8517,B 24.9519,C -1.6019,E1 24.8398,E2 269.3322} C_DIS
LIN {X -120.3819,Y 1.0027,Z 126,A 175.3773,B 24.9519,C -1.6037,E1 24.8398,E2 270.811} C_DIS
LIN {X -120.3207,Y 3.9591,Z 126,A 173.9202,B 24.9517,C -1.6062,E1 24.8399,E2 272.2709} C_DIS
LIN {X -120.1344,Y 7.7792,Z 126,A 172.0084,B 24.9515,C -1.6083,E1 24.8402,E2 274.1892} C_DIS
LIN {X -119.8124,Y 11.7535,Z 126,A 169.9928,B 24.9515,C -1.6096,E1 24.8407,E2 276.2139} C_DIS
LIN {X -119.3004,Y 16.1413,Z 126,A 167.8025,B 24.9513,C -1.6128,E1 24.8415,E2 278.4097} C_DIS
LIN {X -118.7238,Y 19.9333,Z 126,A 166.2528,B 24.9502,C -1.6303,E1 24.8422,E2 279.9268} C_DIS
LIN {X -118.1463,Y 23.1142,Z 126,A 164.5627,B 24.9502,C -1.6289,E1 24.8431,E2 281.6303} C_DIS
LIN {X -117.136,Y 27.7913,Z 126,A 162.4162,B 24.9495,C -1.6417,E1 24.8444,E2 283.7588} C_DIS
LIN {X -116.3761,Y 30.8163,Z 126,A 160.3604,B 24.9507,C -1.6226,E1 24.8459,E2 285.8722} C_DIS
LIN {X -115.2799,Y 34.6906,Z 126,A 159.1328,B 24.9485,C -1.6576,E1 24.8468,E2 287.0235} C_DIS
LIN {X -111.8674,Y 44.4815,Z 126,A 154.0512,B 24.9479,C -1.6669,E1 24.8515,E2 292.1118} C_DIS
LIN {X -110.8158,Y 47.0385,Z 126,A 152.7009,B 24.9478,C -1.6695,E1 24.8529,E2 293.4634} C_DIS
LIN {X -109.3887,Y 50.2707,Z 126,A 150.9446,B 24.9476,C -1.6715,E1 24.855,E2 295.2245} C_DIS
LIN {X -107.4938,Y 54.205,Z 126,A 148.9491,B 24.947,C -1.6812,E1 24.8574,E2 297.2076} C_DIS
LIN {X -104.0185,Y 60.6074,Z 126,A 145.4193,B 24.9466,C -1.6888,E1 24.8622,E2 300.738} C_DIS
LIN {X -102.0455,Y 63.8702,Z 126,A 143.5384,B 24.9464,C -1.6912,E1 24.8649,E2 302.6226} C_DIS
LIN {X -100.01,Y 67.015,Z 126,A 141.748,B 24.9461,C -1.696,E1 24.8676,E2 304.4108} C_DIS
LIN {X -97.831,Y 70.156,Z 126,A 139.1295,B 24.9479,C -1.6674,E1 24.872,E2 307.1101} C_DIS
LIN {X -94.6078,Y 74.4453,Z 126,A 137.6116,B 24.9447,C -1.718,E1 24.8744,E2 308.5146} C_DIS
LIN {X -91.4473,Y 78.2953,Z 126,A 135.0456,B 24.9448,C -1.7159,E1 24.879,E2 311.0975} C_DIS
LIN {X -89.6245,Y 80.3749,Z 126,A 133.6382,B 24.9448,C -1.7154,E1 24.8816,E2 312.5123} C_DIS
LIN {X -86.9373,Y 83.2749,Z 126,A 131.961,B 24.944,C -1.7289,E1 24.8848,E2 314.1649} C_DIS
LIN {X -84.8267,Y 85.4237,Z 126,A 130.2265,B 24.9446,C -1.7195,E1 24.8883,E2 315.929} C_DIS
LIN {X -81.9101,Y 88.2264,Z 126,A 128.2786,B 24.9444,C -1.7231,E1 24.8922,E2 317.8763} C_DIS
LIN {X -79.2777,Y 90.5966,Z 126,A 126.6239,B 24.944,C -1.7284,E1 24.8956,E2 319.5251} C_DIS
LIN {X -76.9206,Y 92.6062,Z 126,A 125.1832,B 24.9437,C -1.7332,E1 24.8987,E2 320.96} C_DIS
LIN {X -73.4336,Y 95.3949,Z 126,A 123.0927,B 24.9433,C -1.7393,E1 24.9033,E2 323.0437} C_DIS
LIN {X -70.595,Y 97.5164,Z 126,A 121.031,B 24.9441,C -1.7266,E1 24.908,E2 325.1428} C_DIS
LIN {X -67.9391,Y 99.3843,Z 126,A 119.9576,B 24.9426,C -1.7501,E1 24.9104,E2 326.164} C_DIS
LIN {X -65.278,Y 101.1511,Z 126,A 118.2882,B 24.9428,C -1.7466,E1 24.9143,E2 327.8471} C_DIS
LIN {X -61.9321,Y 103.2355,Z 126,A 116.228,B 24.9431,C -1.7421,E1 24.9192,E2 329.9243} C_DIS
LIN {X -58.3487,Y 105.3008,Z 126,A 114.3702,B 24.9426,C -1.7504,E1 24.9237,E2 331.7679} C_DIS
LIN {X -54.8326,Y 107.1731,Z 126,A 112.5118,B 24.9423,C -1.7553,E1 24.9283,E2 333.6198} C_DIS
LIN {X -51.3574,Y 108.8828,Z 126,A 110.2322,B 24.9433,C -1.7392,E1 24.9342,E2 335.9434} C_DIS
LIN {X -47.9941,Y 110.405,Z 126,A 108.9144,B 24.9419,C -1.761,E1 24.9374,E2 337.2126} C_DIS
LIN {X -44.9176,Y 111.6931,Z 126,A 107.0751,B 24.9425,C -1.7522,E1 24.9422,E2 339.077} C_DIS
LIN {X -40.2061,Y 113.4737,Z 126,A 104.903,B 24.9416,C -1.7652,E1 24.9479,E2 341.2225} C_DIS
LIN {X -37.0789,Y 114.5331,Z 126,A 103.3717,B 24.9414,C -1.7689,E1 24.9519,E2 342.7479} C_DIS
LIN {X -33.9027,Y 115.5137,Z 126,A 101.8056,B 24.9412,C -1.7714,E1 24.9561,E2 344.3108} C_DIS
LIN {X -30.6806,Y 116.4121,Z 126,A 100.0786,B 24.9415,C -1.767,E1 24.9608,E2 346.0507} C_DIS
LIN {X -27.1815,Y 117.2768,Z 126,A 98.45,B 24.9411,C -1.7725,E1 24.9652,E2 347.6684} C_DIS
LIN {X -23.7013,Y 118.0305,Z 126,A 96.8149,B 24.9408,C -1.7766,E1 24.9696,E2 349.2958} C_DIS
LIN {X -21.2437,Y 118.4964,Z 126,A 95.6199,B 24.9408,C -1.7774,E1 24.9729,E2 350.4903} C_DIS
LIN {X -18.2147,Y 118.9997,Z 126,A 94.1164,B 24.9408,C -1.7765,E1 24.977,E2 351.9971} C_DIS
LIN {X -14.4912,Y 119.5112,Z 126,A 92.2206,B 24.9411,C -1.7728,E1 24.9823,E2 353.9032} C_DIS
LIN {X -11.0459,Y 119.8777,Z 126,A 90.6653,B 24.9408,C -1.7779,E1 24.9866,E2 355.4472} C_DIS
LIN {X -7.9171,Y 120.1251,Z 126,A 89.1441,B 24.9408,C -1.7773,E1 24.9909,E2 356.9705} C_DIS
LIN {X -3.8827,Y 120.3231,Z 126,A 87.2744,B 24.9406,C -1.7803,E1 24.996,E2 358.8335} C_DIS
LIN {X -0.7163,Y 120.3834,Z 126,A 85.3272,B 24.9419,C -1.7609,E1 25.0016,E2 360.8267} C_DIS
LIN {X 2.9431,Y 120.3513,Z 126,A 84.048,B 24.9405,C -1.7819,E1 25.0051,E2 362.0558} C_DIS
LIN {X 6.4127,Y 120.2148,Z 126,A 82.2753,B 24.9408,C -1.7766,E1 25.01,E2 363.8407} C_DIS
LIN {X 10.4694,Y 119.9309,Z 126,A 79.8978,B 24.9422,C -1.7564,E1 25.0168,E2 366.2646} C_DIS
LIN {X 14.4097,Y 119.5207,Z 126,A 78.6902,B 24.9402,C -1.7869,E1 25.0199,E2 367.3992} C_DIS
LIN {X 17.1075,Y 119.1639,Z 126,A 77.2627,B 24.9406,C -1.7805,E1 25.0239,E2 368.8406} C_DIS
LIN {X 19.9105,Y 118.7276,Z 126,A 75.8719,B 24.9407,C -1.7782,E1 25.0278,E2 370.2355} C_DIS
LIN {X 23.7715,Y 118.0161,Z 126,A 73.9588,B 24.9409,C -1.7754,E1 25.033,E2 372.1531} C_DIS
LIN {X 26.9773,Y 117.324,Z 126,A 72.4254,B 24.9409,C -1.7758,E1 25.0372,E2 373.6833} C_DIS
LIN {X 30.0977,Y 116.5625,Z 126,A 70.9009,B 24.9409,C -1.7751,E1 25.0413,E2 375.2073} C_DIS
LIN {X 33.6825,Y 115.579,Z 126,A 68.9604,B 24.9416,C -1.7659,E1 25.0466,E2 377.1662} C_DIS
LIN {X 37.1539,Y 114.5088,Z 126,A 67.4195,B 24.9411,C -1.7733,E1 25.0506,E2 378.687} C_DIS
LIN {X 40.5599,Y 113.3495,Z 126,A 65.7614,B 24.9411,C -1.7742,E1 25.055,E2 380.3395} C_DIS
LIN {X 43.56,Y 112.2294,Z 126,A 63.6692,B 24.9428,C -1.7465,E1 25.0606,E2 382.4928} C_DIS
LIN {X 47.4455,Y 110.6441,Z 126,A 62.2515,B 24.9412,C -1.7711,E1 25.0641,E2 383.8488} C_DIS
LIN {X 51.4088,Y 108.8589,Z 126,A 60.2097,B 24.9412,C -1.7699,E1 25.0693,E2 385.8883} C_DIS
LIN {X 55.3958,Y 106.8852,Z 126,A 58.0786,B 24.9415,C -1.7666,E1 25.0746,E2 388.0215} C_DIS
LIN {X 58.2291,Y 105.3676,Z 126,A 56.3838,B 24.9422,C -1.7567,E1 25.0788,E2 389.7348} C_DIS
LIN {X 61.3049,Y 103.6069,Z 126,A 54.6324,B 24.9425,C -1.7512,E1 25.083,E2 391.4938} C_DIS
LIN {X 64.0981,Y 101.9031,Z 126,A 53.1455,B 24.9425,C -1.7521,E1 25.0865,E2 392.974} C_DIS
LIN {X 67.8901,Y 99.4175,Z 126,A 51.1069,B 24.9423,C -1.7541,E1 25.0912,E2 395.0009} C_DIS
LIN {X 71.0168,Y 97.2075,Z 126,A 49.2772,B 24.9426,C -1.7506,E1 25.0954,E2 396.8325} C_DIS
LIN {X 74.2672,Y 94.7486,Z 126,A 47.3031,B 24.9429,C -1.7454,E1 25.0998,E2 398.8117} C_DIS
LIN {X 77.422,Y 92.1895,Z 126,A 45.5256,B 24.9427,C -1.7491,E1 25.1036,E2 400.5737} C_DIS
LIN {X 79.5335,Y 90.3732,Z 126,A 44.1692,B 24.9429,C -1.745,E1 25.1064,E2 401.9343} C_DIS
LIN {X 81.839,Y 88.2917,Z 126,A 42.5792,B 24.9435,C -1.7366,E1 25.1097,E2 403.5377} C_DIS
LIN {X 84.4936,Y 85.7527,Z 126,A 40.9189,B 24.9435,C -1.7371,E1 25.1131,E2 405.1899} C_DIS
LIN {X 86.988,Y 83.2224,Z 126,A 39.2583,B 24.9435,C -1.7349,E1 25.1163,E2 406.8488} C_DIS
LIN {X 89.4198,Y 80.6036,Z 126,A 37.5019,B 24.944,C -1.7283,E1 25.1196,E2 408.6128} C_DIS
LIN {X 91.6499,Y 78.0575,Z 126,A 36.0028,B 24.944,C -1.73,E1 25.1223,E2 410.1014} C_DIS
LIN {X 93.8672,Y 75.3786,Z 126,A 34.2618,B 24.9444,C -1.7218,E1 25.1254,E2 411.8534} C_DIS
LIN {X 96.1604,Y 72.4284,Z 126,A 32.479,B 24.9447,C -1.7172,E1 25.1285,E2 413.6386} C_DIS
LIN {X 98.3385,Y 69.4446,Z 126,A 30.6666,B 24.9452,C -1.7101,E1 25.1314,E2 415.459} C_DIS
LIN {X 100.602,Y 66.1207,Z 126,A 28.8956,B 24.9451,C -1.7121,E1 25.1342,E2 417.2166} C_DIS
LIN {X 102.3542,Y 63.376,Z 126,A 27.3526,B 24.9453,C -1.7083,E1 25.1365,E2 418.7608} C_DIS
LIN {X 103.9858,Y 60.6639,Z 126,A 25.4576,B 24.9468,C -1.6854,E1 25.1392,E2 420.7} C_DIS
LIN {X 105.6171,Y 57.7744,Z 126,A 24.2336,B 24.946,C -1.6982,E1 25.1408,E2 421.8874} C_DIS
LIN {X 107.3311,Y 54.5233,Z 126,A 22.491,B 24.9462,C -1.6937,E1 25.143,E2 423.6316} C_DIS
LIN {X 109.1939,Y 50.6891,Z 126,A 20.5047,B 24.9465,C -1.6899,E1 25.1454,E2 425.6159} C_DIS
LIN {X 110.7648,Y 47.1598,Z 126,A 18.5028,B 24.9473,C -1.6766,E1 25.1477,E2 427.6383} C_DIS
LIN {X 113.3043,Y 40.6838,Z 126,A 15.4241,B 24.9473,C -1.678,E1 25.1508,E2 430.6965} C_DIS
LIN {X 114.5217,Y 37.1143,Z 126,A 13.5789,B 24.9477,C -1.6702,E1 25.1524,E2 432.5499} C_DIS
LIN {X 115.4026,Y 34.2772,Z 126,A 12.1237,B 24.9481,C -1.6638,E1 25.1536,E2 434.0118} C_DIS
LIN {X 116.7194,Y 29.4874,Z 126,A 9.7266,B 24.9487,C -1.6548,E1 25.1553,E2 436.4163} C_DIS
LIN {X 117.6453,Y 25.5395,Z 126,A 7.9979,B 24.9484,C -1.6586,E1 25.1563,E2 438.1259} C_DIS
LIN {X 118.2379,Y 22.638,Z 126,A 6.5428,B 24.9489,C -1.6519,E1 25.1571,E2 439.5883} C_DIS
LIN {X 118.875,Y 19.0215,Z 126,A 4.6825,B 24.9496,C -1.6408,E1 25.158,E2 441.4639} C_DIS
LIN {X 119.3899,Y 15.4508,Z 126,A 3.0947,B 24.9495,C -1.6417,E1 25.1586,E2 443.0403} C_DIS
LIN {X 119.8195,Y 11.6769,Z 126,A 1.389,B 24.9495,C -1.6408,E1 25.1591,E2 444.7379} C_DIS
LIN {X 120.2718,Y 5.2329,Z 126,A -2.4719,B 24.9525,C -1.5923,E1 25.1597,E2 448.6901} C_DIS
LIN {X 120.3873,Y 0.1334,Z 126,A -4.0989,B 24.9506,C -1.6236,E1 25.1597,E2 450.2339} C_DIS
LIN {X 120.3556,Y -2.7321,Z 126,A -6.0882,B 24.9527,C -1.5884,E1 25.1597,E2 452.2942} C_DIS
LIN {X 120.1816,Y -7.0142,Z 126,A -8.0446,B 24.9529,C -1.5858,E1 25.1593,E2 454.2452} C_DIS
LIN {X 119.8854,Y -10.9626,Z 126,A -9.1089,B 24.9508,C -1.62,E1 25.1591,E2 455.2226} C_DIS
LIN {X 119.3688,Y -15.6137,Z 126,A -11.6504,B 24.9522,C -1.5972,E1 25.1583,E2 457.8029} C_DIS
LIN {X 118.9297,Y -18.6674,Z 126,A -13.151,B 24.9526,C -1.5908,E1 25.1577,E2 459.3097} C_DIS
LIN {X 118.2485,Y -22.5835,Z 126,A -15.0075,B 24.9528,C -1.5863,E1 25.1567,E2 461.1658} C_DIS
LIN {X 117.5432,Y -26.0077,Z 126,A -16.5901,B 24.9529,C -1.5849,E1 25.1558,E2 462.7425} C_DIS
LIN {X 116.6761,Y -29.6557,Z 126,A -18.4611,B 24.9535,C -1.5749,E1 25.1546,E2 464.6262} C_DIS
LIN {X 115.7412,Y -33.1173,Z 126,A -20.0896,B 24.9536,C -1.5733,E1 25.1534,E2 466.2493} C_DIS
LIN {X 114.7173,Y -36.5095,Z 126,A -21.851,B 24.9542,C -1.5642,E1 25.1519,E2 468.022} C_DIS
LIN {X 113.4911,Y -40.1566,Z 126,A -23.5661,B 24.9542,C -1.5642,E1 25.1503,E2 469.7276} C_DIS
LIN {X 112.2458,Y -43.5183,Z 126,A -25.3011,B 24.9546,C -1.5573,E1 25.1486,E2 471.4689} C_DIS
LIN {X 110.6309,Y -47.4759,Z 126,A -27.2381,B 24.9546,C -1.5558,E1 25.1466,E2 473.3989} C_DIS
LIN {X 109.2632,Y -50.5402,Z 126,A -28.9413,B 24.9552,C -1.5457,E1 25.1446,E2 475.1168} C_DIS
LIN {X 107.7481,Y -53.6945,Z 126,A -30.542,B 24.9553,C -1.5438,E1 25.1426,E2 476.7133} C_DIS
LIN {X 106.0405,Y -56.9938,Z 126,A -32.3006,B 24.9556,C -1.539,E1 25.1403,E2 478.4741} C_DIS
LIN {X 104.1614,Y -60.3595,Z 126,A -34.1609,B 24.956,C -1.5323,E1 25.1378,E2 480.3404} C_DIS
LIN {X 101.0899,Y -65.3733,Z 126,A -36.8698,B 24.9562,C -1.5286,E1 25.1338,E2 483.0444} C_DIS
LIN {X 99.5041,Y -67.7622,Z 126,A -38.17,B 24.9562,C -1.5279,E1 25.1317,E2 484.3398} C_DIS
LIN {X 97.9215,Y -70.0291,Z 126,A -39.5782,B 24.9567,C -1.5196,E1 25.1295,E2 485.7605} C_DIS
LIN {X 95.718,Y -73.0142,Z 126,A -41.5237,B 24.9575,C -1.506,E1 25.1262,E2 487.7289} C_DIS
LIN {X 93.0234,Y -76.4184,Z 126,A -44.1943,B 24.9595,C -1.4712,E1 25.1213,E2 490.4692} C_DIS
LIN {X 89.4777,Y -80.5389,Z 126,A -45.9315,B 24.9575,C -1.5056,E1 25.1183,E2 492.1175} C_DIS
LIN {X 85.3278,Y -84.9238,Z 126,A -48.7113,B 24.9577,C -1.5029,E1 25.1129,E2 494.8916} C_DIS
LIN {X 83.4672,Y -86.752,Z 126,A -50.473,B 24.9593,C -1.4747,E1 25.1092,E2 496.7126} C_DIS
LIN {X 80.716,Y -89.3192,Z 126,A -52.6741,B 24.9606,C -1.4508,E1 25.1046,E2 498.9614} C_DIS
LIN {X 76.4228,Y -93.0198,Z 126,A -54.4629,B 24.9585,C -1.4883,E1 25.1009,E2 500.6546} C_DIS
LIN {X 71.7615,Y -96.6613,Z 126,A -57.8705,B 24.9604,C -1.4537,E1 25.0932,E2 504.1316} C_DIS
LIN {X 68.3212,Y -99.1217,Z 126,A -59.1587,B 24.9587,C -1.4844,E1 25.0905,E2 505.3429} C_DIS
LIN {X 66.0537,Y -100.6461,Z 126,A -60.6086,B 24.9593,C -1.4746,E1 25.087,E2 506.8112} C_DIS
LIN {X 62.3404,Y -102.9874,Z 126,A -62.5919,B 24.9593,C -1.4756,E1 25.0824,E2 508.7856} C_DIS
LIN {X 59.7287,Y -104.5239,Z 126,A -64.0923,B 24.9595,C -1.4702,E1 25.0787,E2 510.2943} C_DIS
LIN {X 55.7654,Y -106.6913,Z 126,A -66.2461,B 24.9597,C -1.4662,E1 25.0734,E2 512.4514} C_DIS
LIN {X 52.5705,Y -108.3016,Z 126,A -67.986,B 24.96,C -1.4616,E1 25.069,E2 514.1974} C_DIS
LIN {X 49.2785,Y -109.8378,Z 126,A -69.6818,B 24.96,C -1.4605,E1 25.0647,E2 515.8917} C_DIS
LIN {X 46.1674,Y -111.1829,Z 126,A -71.2382,B 24.96,C -1.4607,E1 25.0608,E2 517.4437} C_DIS
LIN {X 43.3618,Y -112.3062,Z 126,A -73.1796,B 24.9614,C -1.4349,E1 25.0556,E2 519.4419} C_DIS
LIN {X 39.8962,Y -113.5825,Z 126,A -74.8787,B 24.9614,C -1.4354,E1 25.0511,E2 521.1365} C_DIS
LIN {X 36.4701,Y -114.7301,Z 126,A -76.1904,B 24.9605,C -1.4525,E1 25.0477,E2 522.4052} C_DIS
LIN {X 32.5348,Y -115.9062,Z 126,A -78.1781,B 24.9607,C -1.4487,E1 25.0424,E2 524.3985} C_DIS
LIN {X 28.9542,Y -116.8525,Z 126,A -79.9452,B 24.9607,C -1.4467,E1 25.0376,E2 526.1677} C_DIS
LIN {X 25.484,Y -117.6574,Z 126,A -81.6208,B 24.9608,C -1.446,E1 25.033,E2 527.8427} C_DIS
LIN {X 21.5384,Y -118.4434,Z 126,A -83.505,B 24.9608,C -1.4458,E1 25.0279,E2 529.7251} C_DIS
LIN {X 17.6783,Y -119.0827,Z 126,A -85.5419,B 24.9614,C -1.4363,E1 25.0222,E2 531.7827} C_DIS
LIN {X 13.6789,Y -119.6063,Z 126,A -87.394,B 24.9613,C -1.4382,E1 25.0171,E2 533.6287} C_DIS
LIN {X 9.7038,Y -119.9939,Z 126,A -89.7444,B 24.9624,C -1.4165,E1 25.0104,E2 536.0294} C_DIS
LIN {X 5.435,Y -120.2631,Z 126,A -90.9784,B 24.9605,C -1.4528,E1 25.0072,E2 537.177} C_DIS
LIN {X 0.8412,Y -120.3739,Z 126,A -92.351,B 24.9584,C -1.4903,E1 25.0037,E2 538.4602} C_DIS
Enddeposition()
LIN {X 0.8412,Y -120.3739,Z 126,A -92.351,B 24.9584,C -1.4903,E1 25.0037,E2 538.4602} C_DIS
Startdeposition()
$VEL.CP = VEL_PRINT
LIN {X 3.8657,Y -119.4635,Z 126,A -91.6264,B 24.9594,C -1.4715,E1 25.0055,E2 537.7803} C_DIS
LIN {X 7.2676,Y -119.3058,Z 126,A -89.5126,B 24.9582,C -1.4946,E1 25.0116,E2 535.6126} C_DIS
LIN {X 10.8717,Y -119.0304,Z 126,A -87.9162,B 24.9585,C -1.4891,E1 25.016,E2 534.0301} C_DIS
LIN {X 14.1551,Y -118.685,Z 126,A -86.357,B 24.9585,C -1.489,E1 25.0203,E2 532.4723} C_DIS
LIN {X 17.9043,Y -118.1778,Z 126,A -84.4568,B 24.9582,C -1.4943,E1 25.0256,E2 530.5613} C_DIS
LIN {X 21.4539,Y -117.5851,Z 126,A -82.7565,B 24.9582,C -1.4945,E1 25.0302,E2 528.8622} C_DIS
LIN {X 25.3643,Y -116.8036,Z 126,A -80.8829,B 24.9582,C -1.4944,E1 25.0353,E2 526.9912} C_DIS
LIN {X 28.9287,Y -115.9738,Z 126,A -79.0349,B 24.9578,C -1.5006,E1 25.0404,E2 525.1313} C_DIS
LIN {X 32.3699,Y -115.0594,Z 126,A -77.3525,B 24.9578,C -1.5013,E1 25.0449,E2 523.4499} C_DIS
LIN {X 37.7771,Y -113.3997,Z 126,A -74.2719,B 24.9566,C -1.5222,E1 25.0532,E2 520.3255} C_DIS
LIN {X 41.3446,Y -112.1482,Z 126,A -72.6731,B 24.957,C -1.5144,E1 25.0574,E2 518.7486} C_DIS
LIN {X 45.9436,Y -110.3443,Z 126,A -70.4483,B 24.9572,C -1.5109,E1 25.0631,E2 516.537} C_DIS
LIN {X 49.0548,Y -108.9957,Z 126,A -68.9022,B 24.9573,C -1.5096,E1 25.067,E2 514.9978} C_DIS
LIN {X 52.1441,Y -107.5527,Z 126,A -67.3759,B 24.9574,C -1.5071,E1 25.0708,E2 513.4815} C_DIS
LIN {X 55.179,Y -106.0285,Z 126,A -64.8089,B 24.9547,C -1.5554,E1 25.0775,E2 510.8075} C_DIS
LIN {X 60.2382,Y -103.2387,Z 126,A -63.001,B 24.9571,C -1.5136,E1 25.0816,E2 509.1037} C_DIS
LIN {X 63.6193,Y -101.1886,Z 126,A -61.1236,B 24.9569,C -1.5164,E1 25.0861,E2 507.2256} C_DIS
LIN {X 66.0546,Y -99.6158,Z 126,A -59.6414,B 24.9565,C -1.5237,E1 25.0896,E2 505.7312} C_DIS
LIN {X 68.3814,Y -98.0329,Z 126,A -57.9848,B 24.9555,C -1.5414,E1 25.0934,E2 504.0384} C_DIS
LIN {X 71.0448,Y -96.1215,Z 126,A -56.3538,B 24.9551,C -1.5476,E1 25.0971,E2 502.3985} C_DIS
LIN {X 73.806,Y -94.0173,Z 126,A -54.9971,B 24.9558,C -1.5363,E1 25.1,E2 501.0736} C_DIS
LIN {X 76.5889,Y -91.764,Z 126,A -52.744,B 24.954,C -1.5665,E1 25.105,E2 498.7579} C_DIS
LIN {X 80.1426,Y -88.6787,Z 126,A -50.3437,B 24.9533,C -1.5789,E1 25.11,E2 496.3378} C_DIS
LIN {X 84.0075,Y -85.0245,Z 126,A -48.6074,B 24.9553,C -1.5451,E1 25.1133,E2 494.6886} C_DIS
LIN {X 88.8343,Y -79.9687,Z 126,A -44.6931,B 24.9531,C -1.5814,E1 25.1209,E2 490.7059} C_DIS
LIN {X 91.694,Y -76.6732,Z 126,A -43.3914,B 24.9551,C -1.548,E1 25.1231,E2 489.4889} C_DIS
LIN {X 93.0981,Y -74.9621,Z 126,A -42.0655,B 24.9542,C -1.5638,E1 25.1255,E2 488.1318} C_DIS
LIN {X 95.3024,Y -72.1392,Z 126,A -40.5986,B 24.9546,C -1.5562,E1 25.1279,E2 486.6897} C_DIS
LIN {X 96.7597,Y -70.1732,Z 126,A -39.1896,B 24.9538,C -1.5711,E1 25.1303,E2 485.2526} C_DIS
LIN {X 99.4862,Y -66.2512,Z 126,A -36.9389,B 24.9535,C -1.5756,E1 25.1338,E2 483.0022} C_DIS
LIN {X 102.3241,Y -61.7764,Z 126,A -34.5381,B 24.9535,C -1.5761,E1 25.1374,E2 480.6125} C_DIS
LIN {X 103.7897,Y -59.2808,Z 126,A -32.884,B 24.9524,C -1.5934,E1 25.1397,E2 478.9262} C_DIS
LIN {X 105.5811,Y -56.0285,Z 126,A -31.2655,B 24.9526,C -1.5907,E1 25.1418,E2 477.3225} C_DIS
LIN {X 107.1567,Y -52.9517,Z 126,A -29.6416,B 24.9524,C -1.5941,E1 25.1439,E2 475.6992} C_DIS
LIN {X 108.8554,Y -49.3661,Z 126,A -27.2073,B 24.9504,C -1.6264,E1 25.1468,E2 473.202} C_DIS
LIN {X 110.5753,Y -45.3833,Z 126,A -25.921,B 24.9524,C -1.5934,E1 25.1481,E2 472.0005} C_DIS
LIN {X 111.596,Y -42.8138,Z 126,A -24.2543,B 24.9512,C -1.6144,E1 25.1498,E2 470.2934} C_DIS
LIN {X 112.8917,Y -39.2683,Z 126,A -22.6232,B 24.9514,C -1.6113,E1 25.1513,E2 468.6789} C_DIS
LIN {X 114.0245,Y -35.8478,Z 126,A -20.8428,B 24.9509,C -1.6194,E1 25.1528,E2 466.8894} C_DIS
LIN {X 114.9714,Y -32.6804,Z 126,A -19.2563,B 24.9505,C -1.6246,E1 25.1541,E2 465.2998} C_DIS
LIN {X 116.1813,Y -28.0783,Z 126,A -17.0812,B 24.9505,C -1.6267,E1 25.1556,E2 463.1323} C_DIS
LIN {X 116.9364,Y -24.7556,Z 126,A -15.2991,B 24.9496,C -1.6393,E1 25.1566,E2 461.3308} C_DIS
LIN {X 117.6629,Y -21.0211,Z 126,A -13.6097,B 24.9496,C -1.6386,E1 25.1575,E2 459.6529} C_DIS
LIN {X 118.287,Y -17.168,Z 126,A -11.7056,B 24.9492,C -1.6464,E1 25.1583,E2 457.7417} C_DIS
LIN {X 118.7447,Y -13.6453,Z 126,A -10.1159,B 24.9492,C -1.6464,E1 25.1589,E2 456.1615} C_DIS
LIN {X 119.0819,Y -10.3146,Z 126,A -8.2879,B 24.9482,C -1.6626,E1 25.1593,E2 454.3059} C_DIS
LIN {X 119.3919,Y -5.6828,Z 126,A -5.8827,B 24.9472,C -1.6789,E1 25.1597,E2 451.8767} C_DIS
LIN {X 119.5027,Y -2.3573,Z 126,A -4.6724,B 24.948,C -1.665,E1 25.1597,E2 450.7063} C_DIS
LIN {X 119.5211,Y 1.1656,Z 126,A -2.4308,B 24.946,C -1.698,E1 25.1597,E2 448.4002} C_DIS
LIN {X 119.4025,Y 5.4361,Z 126,A -0.375,B 24.9455,C -1.7051,E1 25.1595,E2 446.34} C_DIS
LIN {X 119.1212,Y 9.8316,Z 126,A 1.1152,B 24.947,C -1.6811,E1 25.1592,E2 444.9153} C_DIS
LIN {X 118.7447,Y 13.6453,Z 126,A 2.9468,B 24.9467,C -1.6867,E1 25.1586,E2 443.0813} C_DIS
LIN {X 118.3402,Y 16.7933,Z 126,A 4.4563,B 24.9464,C -1.691,E1 25.158,E2 441.5705} C_DIS
LIN {X 117.8536,Y 19.9247,Z 126,A 5.943,B 24.9462,C -1.6943,E1 25.1574,E2 440.0849} C_DIS
LIN {X 117.3301,Y 22.8059,Z 126,A 7.3724,B 24.9458,C -1.7,E1 25.1566,E2 438.6503} C_DIS
LIN {X 116.5171,Y 26.6505,Z 126,A 9.2703,B 24.9454,C -1.7066,E1 25.1555,E2 436.7478} C_DIS
LIN {X 115.6978,Y 30.0085,Z 126,A 10.8969,B 24.9452,C -1.7103,E1 25.1544,E2 435.1219} C_DIS
LIN {X 114.1629,Y 35.4014,Z 126,A 13.2525,B 24.9457,C -1.7022,E1 25.1526,E2 432.7988} C_DIS
LIN {X 113.3628,Y 37.8868,Z 126,A 14.8685,B 24.9443,C -1.7239,E1 25.1511,E2 431.1408} C_DIS
LIN {X 111.6183,Y 42.7539,Z 126,A 17.3937,B 24.9437,C -1.7336,E1 25.1487,E2 428.6069} C_DIS
LIN {X 110.2794,Y 46.0977,Z 126,A 18.9763,B 24.9438,C -1.7316,E1 25.147,E2 427.0377} C_DIS
LIN {X 108.9754,Y 49.0998,Z 126,A 20.5073,B 24.9436,C -1.7343,E1 25.1453,E2 425.5086} C_DIS
LIN {X 107.6719,Y 51.8961,Z 126,A 22.0355,B 24.9432,C -1.741,E1 25.1435,E2 423.973} C_DIS
LIN {X 105.9182,Y 55.3884,Z 126,A 23.889,B 24.9429,C -1.7453,E1 25.1411,E2 422.1192} C_DIS
LIN {X 103.1922,Y 60.3168,Z 126,A 26.4485,B 24.9429,C -1.7458,E1 25.1376,E2 419.5718} C_DIS
LIN {X 100.4837,Y 64.7262,Z 126,A 29.0407,B 24.9421,C -1.7579,E1 25.1338,E2 416.9642} C_DIS
LIN {X 98.1063,Y 68.2758,Z 126,A 30.9303,B 24.9422,C -1.7555,E1 25.1308,E2 415.0896} C_DIS
LIN {X 96.2909,Y 70.8135,Z 126,A 32.5109,B 24.9417,C -1.7634,E1 25.1282,E2 413.498} C_DIS
LIN {X 94.1275,Y 73.6666,Z 126,A 34.6885,B 24.9399,C -1.79,E1 25.1244,E2 411.2679} C_DIS
LIN {X 91.8777,Y 76.4521,Z 126,A 35.9774,B 24.9411,C -1.7733,E1 25.1222,E2 410.0242} C_DIS
LIN {X 89.3904,Y 79.3475,Z 126,A 37.8607,B 24.9406,C -1.7802,E1 25.1187,E2 408.1333} C_DIS
LIN {X 86.8038,Y 82.1686,Z 126,A 39.5671,B 24.9407,C -1.7781,E1 25.1155,E2 406.4392} C_DIS
LIN {X 84.5191,Y 84.5191,Z 126,A 41.3066,B 24.94,C -1.7896,E1 25.112,E2 404.68} C_DIS
LIN {X 81.8108,Y 87.1403,Z 126,A 42.9808,B 24.9401,C -1.7871,E1 25.1087,E2 403.0186} C_DIS
LIN {X 78.9288,Y 89.7598,Z 126,A 44.7975,B 24.9401,C -1.7885,E1 25.1049,E2 401.2059} C_DIS
LIN {X 76.4545,Y 91.8757,Z 126,A 46.5725,B 24.9392,C -1.8018,E1 25.1011,E2 399.4063} C_DIS
LIN {X 73.1394,Y 94.5363,Z 126,A 48.4392,B 24.9394,C -1.7974,E1 25.097,E2 397.5569} C_DIS
LIN {X 70.3024,Y 96.6651,Z 126,A 50.1668,B 24.9392,C -1.8017,E1 25.0931,E2 395.8253} C_DIS
LIN {X 65.8563,Y 99.7465,Z 126,A 52.7102,B 24.939,C -1.8037,E1 25.0873,E2 393.2859} C_DIS
LIN {X 62.8177,Y 101.6894,Z 126,A 54.666,B 24.9381,C -1.8171,E1 25.0826,E2 391.3045} C_DIS
LIN {X 59.7915,Y 103.4963,Z 126,A 56.2783,B 24.9381,C -1.816,E1 25.0787,E2 389.6999} C_DIS
LIN {X 55.6942,Y 105.7572,Z 126,A 58.356,B 24.9385,C -1.8112,E1 25.0736,E2 387.6394} C_DIS
LIN {X 52.3472,Y 107.4552,Z 126,A 60.4602,B 24.9374,C -1.8279,E1 25.0683,E2 385.5014} C_DIS
LIN {X 47.18,Y 109.822,Z 126,A 63.09,B 24.9374,C -1.8265,E1 25.0616,E2 382.8813} C_DIS
LIN {X 43.2959,Y 111.4095,Z 126,A 64.9128,B 24.9379,C -1.8197,E1 25.0569,E2 381.0786} C_DIS
LIN {X 40.4106,Y 112.4889,Z 126,A 66.2653,B 24.9382,C -1.8153,E1 25.0534,E2 379.7394} C_DIS
LIN {X 37.84,Y 113.3786,Z 126,A 67.5904,B 24.9381,C -1.8174,E1 25.0499,E2 378.4119} C_DIS
LIN {X 33.0395,Y 114.8697,Z 126,A 69.9106,B 24.9382,C -1.8151,E1 25.0437,E2 376.1013} C_DIS
LIN {X 29.9566,Y 115.7111,Z 126,A 71.5838,B 24.9377,C -1.8226,E1 25.0392,E2 374.4128} C_DIS
LIN {X 26.7985,Y 116.483,Z 126,A 73.1165,B 24.9377,C -1.8223,E1 25.035,E2 372.8831} C_DIS
LIN {X 23.0053,Y 117.2917,Z 126,A 75.0505,B 24.9375,C -1.8266,E1 25.0297,E2 370.9413} C_DIS
LIN {X 19.6115,Y 117.906,Z 126,A 76.5963,B 24.9378,C -1.8223,E1 25.0255,E2 369.4073} C_DIS
LIN {X 16.4242,Y 118.3927,Z 126,A 78.1583,B 24.9377,C -1.8235,E1 25.0212,E2 367.844} C_DIS
LIN {X 11.9778,Y 118.9251,Z 126,A 80.356,B 24.9375,C -1.8262,E1 25.015,E2 365.6415} C_DIS
LIN {X 8.4628,Y 119.2265,Z 126,A 82.0603,B 24.9375,C -1.8269,E1 25.0103,E2 363.9363} C_DIS
LIN {X 4.0571,Y 119.4576,Z 126,A 83.9416,B 24.9382,C -1.8161,E1 25.0051,E2 362.0811} C_DIS
LIN {X 1.3519,Y 119.5196,Z 126,A 85.5793,B 24.9371,C -1.8314,E1 25.0004,E2 360.4074} C_DIS
LIN {X -2.462,Y 119.5008,Z 126,A 87.2526,B 24.9376,C -1.824,E1 24.9958,E2 358.7517} C_DIS
LIN {X -6.3764,Y 119.3558,Z 126,A 89.1534,B 24.9376,C -1.8244,E1 24.9905,E2 356.8495} C_DIS
LIN {X -9.8645,Y 119.1186,Z 126,A 90.8341,B 24.9376,C -1.8238,E1 24.9858,E2 355.1694} C_DIS
LIN {X -13.7768,Y 118.7293,Z 126,A 92.7103,B 24.9377,C -1.8224,E1 24.9806,E2 353.2954} C_DIS
LIN {X -16.9283,Y 118.321,Z 126,A 94.1889,B 24.9379,C -1.8195,E1 24.9766,E2 351.8227} C_DIS
LIN {X -19.8254,Y 117.8702,Z 126,A 95.5909,B 24.938,C -1.8183,E1 24.9727,E2 350.4222} C_DIS
LIN {X -23.2515,Y 117.2443,Z 126,A 97.4274,B 24.9376,C -1.8244,E1 24.9676,E2 348.5692} C_DIS
LIN {X -27.7991,Y 116.2495,Z 126,A 99.4206,B 24.9385,C -1.8117,E1 24.9623,E2 346.6035} C_DIS
LIN {X -32.918,Y 114.9041,Z 126,A 102.0562,B 24.9384,C -1.8135,E1 24.9551,E2 343.9598} C_DIS
LIN {X -36.5151,Y 113.8119,Z 126,A 103.9507,B 24.9382,C -1.8155,E1 24.9501,E2 342.0572} C_DIS
LIN {X -39.9733,Y 112.6443,Z 126,A 106.3169,B 24.9365,C -1.8407,E1 24.9437,E2 339.6264} C_DIS
LIN {X -44.462,Y 110.9503,Z 126,A 107.8752,B 24.939,C -1.8046,E1 24.9398,E2 338.1505} C_DIS
LIN {X -48.2176,Y 109.3697,Z 126,A 110.1937,B 24.9381,C -1.8178,E1 24.9338,E2 335.7951} C_DIS
LIN {X -54.8257,Y 106.2111,Z 126,A 113.3556,B 24.9395,C -1.7968,E1 24.926,E2 332.675} C_DIS
LIN {X -57.2108,Y 104.9448,Z 126,A 115.4413,B 24.9373,C -1.8293,E1 24.9207,E2 330.506} C_DIS
LIN {X -61.5305,Y 102.4736,Z 126,A 117.3497,B 24.939,C -1.8039,E1 24.9162,E2 328.6522} C_DIS
LIN {X -64.8865,Y 100.3808,Z 126,A 118.9783,B 24.94,C -1.7887,E1 24.9124,E2 327.0547} C_DIS
LIN {X -67.2847,Y 98.7892,Z 126,A 121.204,B 24.9377,C -1.8229,E1 24.9071,E2 324.74} C_DIS
LIN {X -71.5659,Y 95.7331,Z 126,A 122.8695,B 24.9406,C -1.7802,E1 24.9036,E2 323.1703} C_DIS
LIN {X -74.7546,Y 93.2662,Z 126,A 124.8165,B 24.9408,C -1.7766,E1 24.8993,E2 321.2247} C_DIS
LIN {X -77.0657,Y 91.3655,Z 126,A 126.8183,B 24.9394,C -1.798,E1 24.8949,E2 319.1642} C_DIS
LIN {X -79.9337,Y 88.8657,Z 126,A 128.0896,B 24.9413,C -1.7699,E1 24.8924,E2 317.9548} C_DIS
LIN {X -81.954,Y 87.0056,Z 126,A 129.82,B 24.9403,C -1.7846,E1 24.8888,E2 316.1823} C_DIS
LIN {X -84.2559,Y 84.7791,Z 126,A 130.9632,B 24.9417,C -1.764,E1 24.8866,E2 315.0835} C_DIS
LIN {X -86.2995,Y 82.6978,Z 126,A 132.8958,B 24.9404,C -1.7835,E1 24.8827,E2 313.0959} C_DIS
LIN {X -88.8453,Y 79.9564,Z 126,A 134.02,B 24.9426,C -1.7502,E1 24.8808,E2 312.0462} C_DIS
LIN {X -92.6601,Y 75.5026,Z 126,A 137.1005,B 24.9423,C -1.7543,E1 24.8752,E2 308.9418} C_DIS
LIN {X -95.6116,Y 71.7276,Z 126,A 139.4086,B 24.9427,C -1.7485,E1 24.8712,E2 306.6364} C_DIS
LIN {X -98.2515,Y 68.0669,Z 126,A 141.5098,B 24.9433,C -1.7399,E1 24.8678,E2 304.5456} C_DIS
LIN {X -99.9969,Y 65.4766,Z 126,A 142.9959,B 24.9436,C -1.7351,E1 24.8656,E2 303.0632} C_DIS
LIN {X -101.7902,Y 62.6549,Z 126,A 145.1044,B 24.9425,C -1.7521,E1 24.8624,E2 300.9035} C_DIS
LIN {X -103.574,Y 59.6563,Z 126,A 146.6394,B 24.9432,C -1.7414,E1 24.8603,E2 299.3862} C_DIS
LIN {X -106.5244,Y 54.2127,Z 126,A 149.3323,B 24.9445,C -1.7208,E1 24.8568,E2 296.728} C_DIS
LIN {X -108.2191,Y 50.7461,Z 126,A 151.22,B 24.9448,C -1.7168,E1 24.8545,E2 294.8396} C_DIS
LIN {X -109.6235,Y 47.6355,Z 126,A 152.8822,B 24.945,C -1.7129,E1 24.8526,E2 293.1776} C_DIS
LIN {X -111.1558,Y 43.9417,Z 126,A 155.7241,B 24.9428,C -1.7465,E1 24.8496,E2 290.2397} C_DIS
LIN {X -113.206,Y 38.3516,Z 126,A 157.7731,B 24.9456,C -1.703,E1 24.8478,E2 288.2826} C_DIS
LIN {X -114.4365,Y 34.5107,Z 126,A 159.9926,B 24.9453,C -1.709,E1 24.846,E2 286.0361} C_DIS
LIN {X -115.3559,Y 31.2961,Z 126,A 161.2738,B 24.9465,C -1.6902,E1 24.8451,E2 284.7922} C_DIS
LIN {X -116.1361,Y 28.2638,Z 126,A 163.2481,B 24.9455,C -1.7055,E1 24.8437,E2 282.7698} C_DIS
LIN {X -117.026,Y 24.3192,Z 126,A 164.4493,B 24.9479,C -1.668,E1 24.8431,E2 281.6512} C_DIS
LIN {X -117.8082,Y 20.1963,Z 126,A 167.401,B 24.9458,C -1.7014,E1 24.8416,E2 278.6024} C_DIS
LIN {X -118.5206,Y 15.4694,Z 126,A 169.0575,B 24.9479,C -1.6668,E1 24.841,E2 277.0183} C_DIS
LIN {X -118.9614,Y 11.6194,Z 126,A 171.002,B 24.9481,C -1.6644,E1 24.8404,E2 275.0679} C_DIS
LIN {X -119.2628,Y 7.9262,Z 126,A 172.7004,B 24.9487,C -1.6553,E1 24.8401,E2 273.381} C_DIS
LIN {X -119.4616,Y 3.9258,Z 126,A 174.6363,B 24.949,C -1.6497,E1 24.8398,E2 271.4468} C_DIS
LIN {X -119.5253,Y 0.5175,Z 126,A 176.2398,B 24.9494,C -1.6431,E1 24.8398,E2 269.8494} C_DIS
LIN {X -119.5008,Y -2.4595,Z 126,A 177.6662,B 24.9497,C -1.6384,E1 24.8398,E2 268.4255} C_DIS
LIN {X -119.3778,Y -5.9786,Z 126,A 179.5007,B 24.9497,C -1.6391,E1 24.8401,E2 266.5783} C_DIS
LIN {X -119.1411,Y -9.5824,Z 126,A -178.8427,B 24.9502,C -1.6304,E1 24.8404,E2 264.9326} C_DIS
LIN {X -118.8675,Y -12.5278,Z 126,A -177.4258,B 24.9505,C -1.6258,E1 24.8408,E2 263.5183} C_DIS
LIN {X -118.5016,Y -15.6161,Z 126,A -175.9247,B 24.9507,C -1.6214,E1 24.8413,E2 262.0185} C_DIS
LIN {X -117.904,Y -19.6237,Z 126,A -173.6984,B 24.9504,C -1.6273,E1 24.8423,E2 259.765} C_DIS
LIN {X -116.9856,Y -24.5161,Z 126,A -171.6149,B 24.9516,C -1.6068,E1 24.8434,E2 257.718} C_DIS
LIN {X -116.273,Y -27.7025,Z 126,A -169.5499,B 24.9506,C -1.6233,E1 24.8448,E2 255.6016} C_DIS
LIN {X -115.3821,Y -31.1994,Z 126,A -167.9426,B 24.9513,C -1.6127,E1 24.8459,E2 254.0102} C_DIS
LIN {X -113.6266,Y -37.088,Z 126,A -165.2139,B 24.9524,C -1.5944,E1 24.8482,E2 251.3094} C_DIS
LIN {X -112.4486,Y -40.5209,Z 126,A -163.4933,B 24.9527,C -1.5884,E1 24.8498,E2 249.5934} C_DIS
LIN {X -111.1918,Y -43.8501,Z 126,A -161.853,B 24.9532,C -1.5805,E1 24.8514,E2 247.9627} C_DIS
LIN {X -109.8985,Y -47.0015,Z 126,A -159.5487,B 24.9518,C -1.6046,E1 24.854,E2 245.588} C_DIS
LIN {X -108.0192,Y -51.1732,Z 126,A -158.0492,B 24.9539,C -1.5684,E1 24.8557,E2 244.1668} C_DIS
LIN {X -106.0517,Y -55.1349,Z 126,A -155.3411,B 24.9528,C -1.5878,E1 24.8592,E2 241.3979} C_DIS
LIN {X -104.2052,Y -58.5474,Z 126,A -154.0437,B 24.9545,C -1.5584,E1 24.8609,E2 240.1638} C_DIS
LIN {X -102.6171,Y -61.2899,Z 126,A -152.3694,B 24.9543,C -1.561,E1 24.8633,E2 238.4747} C_DIS
LIN {X -97.6117,Y -68.9832,Z 126,A -148.1427,B 24.9555,C -1.5419,E1 24.8698,E2 234.2722} C_DIS
LIN {X -94.9779,Y -72.5663,Z 126,A -146.0198,B 24.9558,C -1.5362,E1 24.8733,E2 232.1527} C_DIS
LIN {X -92.6399,Y -75.5274,Z 126,A -144.0691,B 24.9557,C -1.538,E1 24.8767,E2 230.1885} C_DIS
LIN {X -89.8495,Y -78.8261,Z 126,A -141.977,B 24.9559,C -1.5341,E1 24.8805,E2 228.0962} C_DIS
LIN {X -86.9832,Y -81.9778,Z 126,A -139.8952,B 24.9561,C -1.5312,E1 24.8844,E2 226.0121} C_DIS
LIN {X -83.8199,Y -85.2099,Z 126,A -137.7799,B 24.9565,C -1.5243,E1 24.8886,E2 223.9043} C_DIS
LIN {X -81.3931,Y -87.5331,Z 126,A -136.1684,B 24.9567,C -1.5209,E1 24.8919,E2 222.2942} C_DIS
LIN {X -78.8591,Y -89.8207,Z 126,A -133.8611,B 24.9551,C -1.5474,E1 24.8968,E2 219.9148} C_DIS
LIN {X -75.4134,Y -92.7323,Z 126,A -132.5842,B 24.9576,C -1.504,E1 24.8994,E2 218.7361} C_DIS
LIN {X -72.224,Y -95.2387,Z 126,A -129.9039,B 24.956,C -1.5331,E1 24.9055,E2 215.9771} C_DIS
LIN {X -69.2504,Y -97.421,Z 126,A -128.734,B 24.9577,C -1.5034,E1 24.908,E2 214.8735} C_DIS
LIN {X -67.0027,Y -98.9801,Z 126,A -127.2519,B 24.9573,C -1.5088,E1 24.9114,E2 213.3736} C_DIS
LIN {X -63.6991,Y -101.1388,Z 126,A -125.5385,B 24.958,C -1.4979,E1 24.9154,E2 211.6806} C_DIS
LIN {X -61.9007,Y -102.2486,Z 126,A -124.2552,B 24.9574,C -1.5085,E1 24.9185,E2 210.3684} C_DIS
LIN {X -58.2838,Y -104.3524,Z 126,A -122.3445,B 24.9578,C -1.5014,E1 24.9231,E2 208.4688} C_DIS
LIN {X -55.1078,Y -106.066,Z 126,A -120.2425,B 24.957,C -1.5158,E1 24.9284,E2 206.3268} C_DIS
LIN {X -52.1841,Y -107.5335,Z 126,A -119.1928,B 24.9584,C -1.4905,E1 24.9309,E2 205.3343} C_DIS
LIN {X -47.7141,Y -109.5892,Z 126,A -116.6702,B 24.9581,C -1.4952,E1 24.9374,E2 202.7945} C_DIS
LIN {X -44.1282,Y -111.0826,Z 126,A -114.7732,B 24.9581,C -1.4949,E1 24.9423,E2 200.894} C_DIS
LIN {X -40.8894,Y -112.3142,Z 126,A -113.171,B 24.9584,C -1.4907,E1 24.9465,E2 199.2985} C_DIS
LIN {X -36.1037,Y -113.9451,Z 126,A -110.756,B 24.9585,C -1.4883,E1 24.9529,E2 196.8847} C_DIS
LIN {X -32.4793,Y -115.0284,Z 126,A -108.8993,B 24.9585,C -1.489,E1 24.9579,E2 195.0231} C_DIS
LIN {X -28.8012,Y -116.005,Z 126,A -107.0104,B 24.9584,C -1.4909,E1 24.963,E2 193.1271} C_DIS
LIN {X -25.3992,Y -116.796,Z 126,A -105.4439,B 24.9587,C -1.4852,E1 24.9672,E2 191.5721} C_DIS
LIN {X -22.4568,Y -117.3973,Z 126,A -103.9895,B 24.9587,C -1.4852,E1 24.9712,E2 190.1159} C_DIS
LIN {X -19.4035,Y -117.9408,Z 126,A -102.4729,B 24.9587,C -1.4861,E1 24.9754,E2 188.5957} C_DIS
LIN {X -14.4118,Y -118.6549,Z 126,A -99.9124,B 24.9583,C -1.4922,E1 24.9825,E2 186.0189} C_DIS
LIN {X -10.3673,Y -119.077,Z 126,A -97.5933,B 24.9573,C -1.5093,E1 24.9891,E2 183.6582} C_DIS
LIN {X -6.4851,Y -119.3498,Z 126,A -96.3862,B 24.959,C -1.4788,E1 24.9923,E2 182.523} C_DIS
LIN {X -0.5975,Y -119.5244,Z 126,A -93.4118,B 24.9586,C -1.4861,E1 25.0006,E2 179.5309} C_DIS
LIN {X -0.5975,Y -119.5244,Z 126,A -93.4118,B 24.9586,C -1.4861,E1 25.0006,E2 179.5309} C_DIS
Enddeposition()
LIN {X 0.8396,Y -118.6625,Z 126,A -93.4692,B 24.9597,C -1.467,E1 25.0003,E2 179.6336} C_DIS
Startdeposition()
$VEL.CP = VEL_PRINT
LIN {X -4.6009,Y -118.5779,Z 126,A -96.2368,B 24.9601,C -1.4602,E1 24.9926,E2 182.4176} C_DIS
LIN {X -9.0147,Y -118.3241,Z 126,A -98.2453,B 24.9597,C -1.4659,E1 24.987,E2 184.4134} C_DIS
LIN {X -12.1611,Y -118.0415,Z 126,A -99.604,B 24.9593,C -1.4735,E1 24.9833,E2 185.7546} C_DIS
LIN {X -16.9972,Y -117.4429,Z 126,A -102.1726,B 24.9598,C -1.4642,E1 24.9761,E2 188.3472} C_DIS
LIN {X -20.8439,Y -116.8213,Z 126,A -104.0004,B 24.9597,C -1.4672,E1 24.9711,E2 190.1696} C_DIS
LIN {X -23.8812,Y -116.2383,Z 126,A -105.4344,B 24.9595,C -1.4705,E1 24.9672,E2 191.5974} C_DIS
LIN {X -26.9449,Y -115.5668,Z 126,A -107.0725,B 24.9598,C -1.4657,E1 24.9627,E2 193.249} C_DIS
LIN {X -30.6939,Y -114.6281,Z 126,A -108.9062,B 24.9596,C -1.4683,E1 24.9577,E2 195.0794} C_DIS
LIN {X -34.4416,Y -113.5603,Z 126,A -110.7038,B 24.9593,C -1.4733,E1 24.9529,E2 196.868} C_DIS
LIN {X -39.9525,Y -111.7405,Z 126,A -113.6284,B 24.9595,C -1.4701,E1 24.9452,E2 199.8056} C_DIS
LIN {X -44.581,Y -109.9737,Z 126,A -115.9816,B 24.9593,C -1.4742,E1 24.939,E2 202.1542} C_DIS
LIN {X -48.5453,Y -108.2823,Z 126,A -118.0457,B 24.9591,C -1.4772,E1 24.9338,E2 204.216} C_DIS
LIN {X -51.4229,Y -106.9455,Z 126,A -120.1465,B 24.9604,C -1.4542,E1 24.9283,E2 206.3768} C_DIS
LIN {X -55.2138,Y -105.0385,Z 126,A -121.6905,B 24.959,C -1.4789,E1 24.9246,E2 207.8665} C_DIS
LIN {X -58.8165,Y -103.065,Z 126,A -123.4169,B 24.9583,C -1.4928,E1 24.9205,E2 209.5647} C_DIS
LIN {X -61.3554,Y -101.574,Z 126,A -125.0015,B 24.9585,C -1.4878,E1 24.9166,E2 211.166} C_DIS
LIN {X -64.7233,Y -99.4639,Z 126,A -127.0832,B 24.9588,C -1.4837,E1 24.9117,E2 213.2641} C_DIS
LIN {X -68.3623,Y -96.9986,Z 126,A -129.2024,B 24.9586,C -1.4874,E1 24.9068,E2 215.3818} C_DIS
LIN {X -72.6038,Y -93.8636,Z 126,A -131.851,B 24.9586,C -1.4875,E1 24.9009,E2 218.0395} C_DIS
LIN {X -77.6265,Y -89.7559,Z 126,A -134.8976,B 24.958,C -1.4972,E1 24.8944,E2 221.0747} C_DIS
LIN {X -80.4569,Y -87.2263,Z 126,A -136.9294,B 24.9583,C -1.4925,E1 24.8902,E2 223.126} C_DIS
LIN {X -84.435,Y -83.3809,Z 126,A -139.3163,B 24.9573,C -1.5103,E1 24.8855,E2 225.4805} C_DIS
LIN {X -86.4051,Y -81.3377,Z 126,A -141.0501,B 24.958,C -1.4979,E1 24.8821,E2 227.2514} C_DIS
LIN {X -88.5826,Y -78.961,Z 126,A -142.6239,B 24.9578,C -1.5007,E1 24.8791,E2 228.8256} C_DIS
LIN {X -90.8011,Y -76.4024,Z 126,A -143.98,B 24.9569,C -1.5163,E1 24.8768,E2 230.1507} C_DIS
LIN {X -92.9011,Y -73.8319,Z 126,A -145.5639,B 24.9567,C -1.521,E1 24.874,E2 231.7308} C_DIS
LIN {X -95.7937,Y -70.0372,Z 126,A -147.8618,B 24.9563,C -1.5269,E1 24.8701,E2 234.0256} C_DIS
LIN {X -97.5068,Y -67.632,Z 126,A -150.1717,B 24.9582,C -1.4935,E1 24.8664,E2 236.4264} C_DIS
LIN {X -100.6523,Y -62.8551,Z 126,A -152.0366,B 24.9557,C -1.5383,E1 24.8637,E2 238.1943} C_DIS
LIN {X -102.3765,Y -60.0074,Z 126,A -153.7193,B 24.9557,C -1.5394,E1 24.8613,E2 239.8829} C_DIS
LIN {X -105.9958,Y -53.358,Z 126,A -158.5622,B 24.9578,C -1.5004,E1 24.8549,E2 244.8447} C_DIS
LIN {X -109.0133,Y -46.8838,Z 126,A -160.9008,B 24.9546,C -1.5562,E1 24.8524,E2 247.0631} C_DIS
LIN {X -110.3922,Y -43.5342,Z 126,A -162.6189,B 24.9542,C -1.5627,E1 24.8506,E2 248.7754} C_DIS
LIN {X -111.5006,Y -40.6113,Z 126,A -164.1878,B 24.9542,C -1.5647,E1 24.8491,E2 250.3484} C_DIS
LIN {X -112.8185,Y -36.7929,Z 126,A -165.8202,B 24.953,C -1.5838,E1 24.8476,E2 251.9444} C_DIS
LIN {X -114.2791,Y -31.9702,Z 126,A -168.5223,B 24.9532,C -1.58,E1 24.8455,E2 254.6712} C_DIS
LIN {X -115.6473,Y -26.5962,Z 126,A -171.2122,B 24.9528,C -1.5878,E1 24.8437,E2 257.3582} C_DIS
LIN {X -116.1674,Y -24.2265,Z 126,A -173.0167,B 24.9541,C -1.5654,E1 24.8426,E2 259.2268} C_DIS
LIN {X -117.002,Y -19.805,Z 126,A -174.9981,B 24.9532,C -1.5801,E1 24.8417,E2 261.1848} C_DIS
LIN {X -117.5533,Y -16.2202,Z 126,A -176.391,B 24.952,C -1.6005,E1 24.8411,E2 262.5375} C_DIS
LIN {X -118.0042,Y -12.5176,Z 126,A -178.2613,B 24.9518,C -1.6034,E1 24.8405,E2 264.4119} C_DIS
LIN {X -118.389,Y -8.1052,Z 126,A 179.7647,B 24.951,C -1.6172,E1 24.8401,E2 266.3651} C_DIS
LIN {X -118.5591,Y -5.0402,Z 126,A 178.1849,B 24.951,C -1.6179,E1 24.8399,E2 267.9526} C_DIS
LIN {X -118.6599,Y -1.3905,Z 126,A 176.3626,B 24.9508,C -1.6212,E1 24.8398,E2 269.7781} C_DIS
LIN {X -118.6447,Y 2.2573,Z 126,A 174.6588,B 24.9503,C -1.6293,E1 24.8398,E2 271.4728} C_DIS
LIN {X -118.5271,Y 5.7834,Z 126,A 172.8958,B 24.9501,C -1.6324,E1 24.84,E2 273.239} C_DIS
LIN {X -118.3049,Y 9.2544,Z 126,A 171.1997,B 24.9498,C -1.6372,E1 24.8404,E2 274.9338} C_DIS
LIN {X -117.953,Y 13.0068,Z 126,A 169.4116,B 24.9493,C -1.6445,E1 24.8409,E2 276.7154} C_DIS
LIN {X -116.7698,Y 21.13,Z 126,A 165.4414,B 24.9485,C -1.6571,E1 24.8426,E2 280.6792} C_DIS
LIN {X -115.7849,Y 25.9917,Z 126,A 162.8177,B 24.9486,C -1.6554,E1 24.8441,E2 283.3224} C_DIS
LIN {X -113.9448,Y 33.1454,Z 126,A 159.3131,B 24.9478,C -1.6693,E1 24.8466,E2 286.8141} C_DIS
LIN {X -112.8155,Y 36.8022,Z 126,A 157.8288,B 24.9465,C -1.6903,E1 24.8478,E2 288.257} C_DIS
LIN {X -110.4442,Y 43.4019,Z 126,A 154.1548,B 24.9465,C -1.6889,E1 24.8513,E2 291.9551} C_DIS
LIN {X -109.0112,Y 46.8886,Z 126,A 152.2501,B 24.9465,C -1.691,E1 24.8534,E2 293.8654} C_DIS
LIN {X -107.8182,Y 49.5702,Z 126,A 150.7523,B 24.9464,C -1.692,E1 24.8551,E2 295.369} C_DIS
LIN {X -106.1315,Y 53.0842,Z 126,A 149.0406,B 24.9455,C -1.7047,E1 24.8572,E2 297.0596} C_DIS
LIN {X -103.1841,Y 58.6092,Z 126,A 146.0558,B 24.9449,C -1.7152,E1 24.8612,E2 300.0351} C_DIS
LIN {X -100.7325,Y 62.7267,Z 126,A 143.6261,B 24.9447,C -1.7171,E1 24.8647,E2 302.4728} C_DIS
LIN {X -99.0144,Y 65.4049,Z 126,A 142.2964,B 24.9439,C -1.7301,E1 24.8666,E2 303.7783} C_DIS
LIN {X -96.2222,Y 69.4504,Z 126,A 139.7331,B 24.9439,C -1.7287,E1 24.8708,E2 306.3575} C_DIS
LIN {X -93.2378,Y 73.4059,Z 126,A 137.3192,B 24.9436,C -1.7343,E1 24.8749,E2 308.7696} C_DIS
LIN {X -89.2842,Y 78.1665,Z 126,A 134.5045,B 24.9426,C -1.7494,E1 24.8799,E2 311.5613} C_DIS
LIN {X -85.8935,Y 81.8803,Z 126,A 131.7344,B 24.9432,C -1.7412,E1 24.8852,E2 314.3632} C_DIS
LIN {X -83.5052,Y 84.3123,Z 126,A 129.6895,B 24.944,C -1.7286,E1 24.8893,E2 316.4468} C_DIS
LIN {X -80.6372,Y 87.0609,Z 126,A 127.7174,B 24.9439,C -1.7308,E1 24.8933,E2 318.4215} C_DIS
LIN {X -77.5529,Y 89.8201,Z 126,A 126.1301,B 24.9424,C -1.7526,E1 24.8966,E2 319.9633} C_DIS
LIN {X -74.4548,Y 92.4026,Z 126,A 124.0146,B 24.9426,C -1.7498,E1 24.9012,E2 322.0932} C_DIS
LIN {X -69.7876,Y 95.976,Z 126,A 120.9531,B 24.9428,C -1.7465,E1 24.9081,E2 325.1737} C_DIS
LIN {X -66.6302,Y 98.1941,Z 126,A 119.5383,B 24.9413,C -1.7691,E1 24.9112,E2 326.5394} C_DIS
LIN {X -63.6968,Y 100.1229,Z 126,A 117.5743,B 24.9419,C -1.761,E1 24.9159,E2 328.5291} C_DIS
LIN {X -57.6093,Y 103.7444,Z 126,A 114.3524,B 24.9409,C -1.7756,E1 24.9236,E2 331.7258} C_DIS
LIN {X -55.3782,Y 104.9519,Z 126,A 112.1979,B 24.9434,C -1.7383,E1 24.9292,E2 333.9749} C_DIS
LIN {X -49.7784,Y 107.7213,Z 126,A 110.165,B 24.9403,C -1.7847,E1 24.9341,E2 335.9026} C_DIS
LIN {X -46.4869,Y 109.1825,Z 126,A 108.3492,B 24.9403,C -1.784,E1 24.9387,E2 337.7244} C_DIS
LIN {X -37.4265,Y 112.6107,Z 126,A 103.6322,B 24.9401,C -1.7884,E1 24.9511,E2 342.4406} C_DIS
LIN {X -29.2321,Y 115.0097,Z 126,A 99.7834,B 24.939,C -1.8047,E1 24.9613,E2 346.2568} C_DIS
LIN {X -25.0351,Y 115.9955,Z 126,A 97.4694,B 24.9395,C -1.7965,E1 24.9677,E2 348.5933} C_DIS
LIN {X -21.5075,Y 116.7019,Z 126,A 95.7744,B 24.9393,C -1.7997,E1 24.9723,E2 350.2826} C_DIS
LIN {X -18.3023,Y 117.2464,Z 126,A 94.2947,B 24.9389,C -1.8048,E1 24.9764,E2 351.7516} C_DIS
LIN {X -15.2161,Y 117.6865,Z 126,A 92.65,B 24.9393,C -1.7996,E1 24.9809,E2 353.4099} C_DIS
LIN {X -11.1165,Y 118.1445,Z 126,A 90.6742,B 24.9392,C -1.8014,E1 24.9864,E2 355.3826} C_DIS
LIN {X -7.7093,Y 118.4158,Z 126,A 88.9709,B 24.9392,C -1.7998,E1 24.9912,E2 357.0904} C_DIS
LIN {X -3.9538,Y 118.6007,Z 126,A 87.1757,B 24.9392,C -1.8013,E1 24.9962,E2 358.8824} C_DIS
LIN {X -0.2676,Y 118.6667,Z 126,A 85.0965,B 24.9401,C -1.7884,E1 25.0021,E2 360.9921} C_DIS
LIN {X 3.0607,Y 118.6279,Z 126,A 83.6797,B 24.9395,C -1.797,E1 25.006,E2 362.3882} C_DIS
LIN {X 7.4329,Y 118.4345,Z 126,A 81.7059,B 24.9391,C -1.8033,E1 25.0114,E2 364.3465} C_DIS
LIN {X 10.6423,Y 118.1882,Z 126,A 79.841,B 24.94,C -1.7893,E1 25.0167,E2 366.2435} C_DIS
LIN {X 15.7387,Y 117.6188,Z 126,A 77.586,B 24.9394,C -1.7987,E1 25.0229,E2 368.4746} C_DIS
LIN {X 19.6369,Y 117.0301,Z 126,A 75.807,B 24.939,C -1.8037,E1 25.0278,E2 370.24} C_DIS
LIN {X 23.3991,Y 116.3373,Z 126,A 73.8933,B 24.9393,C -1.7999,E1 25.033,E2 372.1605} C_DIS
LIN {X 26.5361,Y 115.6612,Z 126,A 72.3466,B 24.9393,C -1.7992,E1 25.0372,E2 373.7067} C_DIS
LIN {X 30.5754,Y 114.6601,Z 126,A 70.5925,B 24.9386,C -1.8095,E1 25.0419,E2 375.4337} C_DIS
LIN {X 36.9897,Y 112.7548,Z 126,A 67.146,B 24.9395,C -1.7972,E1 25.0512,E2 378.9032} C_DIS
LIN {X 39.2933,Y 111.9718,Z 126,A 65.702,B 24.9404,C -1.7839,E1 25.0551,E2 380.3757} C_DIS
LIN {X 43.457,Y 110.4226,Z 126,A 63.7078,B 24.94,C -1.7887,E1 25.0602,E2 382.3544} C_DIS
LIN {X 47.0435,Y 108.9437,Z 126,A 62.0293,B 24.9396,C -1.7955,E1 25.0645,E2 384.0127} C_DIS
LIN {X 52.283,Y 106.5287,Z 126,A 59.1656,B 24.94,C -1.7886,E1 25.0718,E2 386.8855} C_DIS
LIN {X 55.3817,Y 104.9501,Z 126,A 57.5895,B 24.9399,C -1.7911,E1 25.0756,E2 388.4513} C_DIS
LIN {X 58.5157,Y 103.2378,Z 126,A 55.8801,B 24.9399,C -1.7893,E1 25.0798,E2 390.1598} C_DIS
LIN {X 62.0358,Y 101.1604,Z 126,A 53.7279,B 24.9407,C -1.7781,E1 25.085,E2 392.3319} C_DIS
LIN {X 65.1038,Y 99.213,Z 126,A 51.4135,B 24.9426,C -1.7495,E1 25.0906,E2 394.7064} C_DIS
LIN {X 69.1001,Y 96.4721,Z 126,A 49.761,B 24.9408,C -1.7772,E1 25.0942,E2 396.2877} C_DIS
LIN {X 72.14,Y 94.2211,Z 126,A 47.5315,B 24.9423,C -1.7552,E1 25.0992,E2 398.5611} C_DIS
LIN {X 74.9715,Y 91.9839,Z 126,A 46.1163,B 24.9415,C -1.7671,E1 25.1022,E2 399.9428} C_DIS
LIN {X 77.9678,Y 89.4577,Z 126,A 44.1661,B 24.9419,C -1.7606,E1 25.1064,E2 401.9007} C_DIS
LIN {X 81.1817,Y 86.5518,Z 126,A 42.1855,B 24.9419,C -1.7615,E1 25.1104,E2 403.8711} C_DIS
LIN {X 83.9112,Y 83.9112,Z 126,A 40.1658,B 24.9427,C -1.7488,E1 25.1145,E2 405.9123} C_DIS
LIN {X 87.1841,Y 80.5029,Z 126,A 38.0304,B 24.9426,C -1.7506,E1 25.1185,E2 408.0341} C_DIS
LIN {X 89.8567,Y 77.5109,Z 126,A 36.0849,B 24.9429,C -1.7457,E1 25.1221,E2 409.9826} C_DIS
LIN {X 94.3042,Y 72.0321,Z 126,A 32.7457,B 24.9432,C -1.7406,E1 25.1279,E2 413.318} C_DIS
LIN {X 96.2506,Y 69.4105,Z 126,A 30.8346,B 24.9445,C -1.7208,E1 25.1311,E2 415.2667} C_DIS
LIN {X 98.2984,Y 66.4761,Z 126,A 29.5595,B 24.9434,C -1.7378,E1 25.1331,E2 416.4953} C_DIS
LIN {X 100.4049,Y 63.2511,Z 126,A 27.8654,B 24.9432,C -1.7408,E1 25.1356,E2 418.174} C_DIS
LIN {X 102.0107,Y 60.6263,Z 126,A 26.1311,B 24.9442,C -1.7249,E1 25.1381,E2 419.9368} C_DIS
LIN {X 104.6121,Y 56.0211,Z 126,A 23.5935,B 24.9446,C -1.7186,E1 25.1416,E2 422.476} C_DIS
LIN {X 106.1661,Y 53.0144,Z 126,A 22.0048,B 24.9448,C -1.7162,E1 25.1436,E2 424.0619} C_DIS
LIN {X 107.707,Y 49.809,Z 126,A 20.2693,B 24.9452,C -1.7104,E1 25.1456,E2 425.8017} C_DIS
LIN {X 109.2377,Y 46.3559,Z 126,A 18.4846,B 24.9454,C -1.707,E1 25.1476,E2 427.5848} C_DIS
LIN {X 111.4876,Y 40.6469,Z 126,A 15.4872,B 24.9461,C -1.6965,E1 25.1506,E2 430.5902} C_DIS
LIN {X 112.7479,Y 37.0111,Z 126,A 12.9106,B 24.9486,C -1.6565,E1 25.153,E2 433.2464} C_DIS
Enddeposition()
END
